gfCNCPoint2[21603] = {X 522.5718, Y 34.1930, Z -3.0000, A 0.000, B 0.000, C 0.000 }
gfCNCPoint2[21604] = {X 522.0666, Y 33.3891, Z -3.0000, A 0.000, B 0.000, C 0.000 }
gfCNCPoint2[21605] = {X 521.7531, Y 32.4929, Z -3.0000, A 0.000, B 0.000, C 0.000 }
gfCNCPoint2[21606] = {X 521.6468, Y 31.5495, Z -3.0000, A 0.000, B 0.000, C 0.000 }
gfCNCPoint2[21607] = {X 521.6468, Y 24.5714, Z -3.0000, A 0.000, B 0.000, C 0.000 }
gfCNCPoint2[21608] = {X 521.7519, Y 23.6330, Z -3.0000, A 0.000, B 0.000, C 0.000 }
gfCNCPoint2[21609] = {X 522.0622, Y 22.7411, Z -3.0000, A 0.000, B 0.000, C 0.000 }
gfCNCPoint2[21610] = {X 522.5621, Y 21.9400, Z -3.0000, A 0.000, B 0.000, C 0.000 }
gfCNCPoint2[21611] = {X 523.2270, Y 21.2694, Z -3.0000, A 0.000, B 0.000, C 0.000 }
gfCNCPoint2[21612] = {X 524.0238, Y 20.7626, Z -3.0000, A 0.000, B 0.000, C 0.000 }
gfCNCPoint2[21613] = {X 524.9130, Y 20.4448, Z -3.0000, A 0.000, B 0.000, C 0.000 }
gfCNCPoint2[21614] = {X 525.8505, Y 20.3316, Z -3.0000, A 0.000, B 0.000, C 0.000 }
gfCNCPoint2[21615] = {X 526.5687, Y 20.3316, Z -3.0000, A 0.000, B 0.000, C 0.000 }
gfCNCPoint2[21616] = {X 527.3869, Y 20.4192, Z -3.0000, A 0.000, B 0.000, C 0.000 }
gfCNCPoint2[21617] = {X 528.1727, Y 20.6632, Z -3.0000, A 0.000, B 0.000, C 0.000 }
gfCNCPoint2[21618] = {X 528.8966, Y 21.0544, Z -3.0000, A 0.000, B 0.000, C 0.000 }
gfCNCPoint2[21619] = {X 529.5313, Y 21.5780, Z -3.0000, A 0.000, B 0.000, C 0.000 }
gfCNCPoint2[21620] = {X 530.0529, Y 22.2144, Z -3.0000, A 0.000, B 0.000, C 0.000 }
gfCNCPoint2[21621] = {X 534.7119, Y 22.2147, Z -3.0000, A 0.000, B 0.000, C 0.000 }
gfCNCPoint2[21622] = {X 534.7119, Y 19.6214, Z -3.0000, A 0.000, B 0.000, C 0.000 }
gfCNCPoint2[21623] = {X 524.1494, Y 19.6210, Z -3.0000, A 0.000, B 0.000, C 0.000 }
gfCNCPoint2[21624] = {X 524.1262, Y 19.6563, Z -3.0000, A 0.000, B 0.000, C 0.000 }
gfCNCPoint2[21625] = {X 523.6036, Y 20.2891, Z -3.0000, A 0.000, B 0.000, C 0.000 }
gfCNCPoint2[21626] = {X 522.9689, Y 20.8095, Z -3.0000, A 0.000, B 0.000, C 0.000 }
gfCNCPoint2[21627] = {X 522.2458, Y 21.1978, Z -3.0000, A 0.000, B 0.000, C 0.000 }
gfCNCPoint2[21628] = {X 521.4615, Y 21.4395, Z -3.0000, A 0.000, B 0.000, C 0.000 }
gfCNCPoint2[21629] = {X 520.6453, Y 21.5256, Z -3.0000, A 0.000, B 0.000, C 0.000 }
gfCNCPoint2[21630] = {X 519.9691, Y 21.5257, Z -3.0000, A 0.000, B 0.000, C 0.000 }
gfCNCPoint2[21631] = {X 519.0256, Y 21.4194, Z -3.0000, A 0.000, B 0.000, C 0.000 }
gfCNCPoint2[21632] = {X 518.1294, Y 21.1058, Z -3.0000, A 0.000, B 0.000, C 0.000 }
gfCNCPoint2[21633] = {X 517.3255, Y 20.6007, Z -3.0000, A 0.000, B 0.000, C 0.000 }
gfCNCPoint2[21634] = {X 516.6541, Y 19.9293, Z -3.0000, A 0.000, B 0.000, C 0.000 }
gfCNCPoint2[21635] = {X 516.1490, Y 19.1254, Z -3.0000, A 0.000, B 0.000, C 0.000 }
gfCNCPoint2[21636] = {X 515.8354, Y 18.2292, Z -3.0000, A 0.000, B 0.000, C 0.000 }
gfCNCPoint2[21637] = {X 515.7291, Y 17.2857, Z -3.0000, A 0.000, B 0.000, C 0.000 }
gfCNCPoint2[21638] = {X 515.7291, Y 10.3077, Z -3.0000, A 0.000, B 0.000, C 0.000 }
gfCNCPoint2[21639] = {X 515.8342, Y 9.3696, Z -3.0000, A 0.000, B 0.000, C 0.000 }
gfCNCPoint2[21640] = {X 516.1442, Y 8.4780, Z -3.0000, A 0.000, B 0.000, C 0.000 }
gfCNCPoint2[21641] = {X 516.6438, Y 7.6771, Z -3.0000, A 0.000, B 0.000, C 0.000 }
gfCNCPoint2[21642] = {X 517.3082, Y 7.0066, Z -3.0000, A 0.000, B 0.000, C 0.000 }
gfCNCPoint2[21643] = {X 518.1045, Y 6.4997, Z -3.0000, A 0.000, B 0.000, C 0.000 }
gfCNCPoint2[21644] = {X 518.9932, Y 6.1815, Z -3.0000, A 0.000, B 0.000, C 0.000 }
gfCNCPoint2[21645] = {X 519.9303, Y 6.0679, Z -3.0000, A 0.000, B 0.000, C 0.000 }
gfCNCPoint2[21646] = {X 520.6494, Y 6.0679, Z -3.0000, A 0.000, B 0.000, C 0.000 }
gfCNCPoint2[21647] = {X 521.4680, Y 6.1552, Z -3.0000, A 0.000, B 0.000, C 0.000 }
gfCNCPoint2[21648] = {X 522.2542, Y 6.3991, Z -3.0000, A 0.000, B 0.000, C 0.000 }
gfCNCPoint2[21649] = {X 522.9784, Y 6.7903, Z -3.0000, A 0.000, B 0.000, C 0.000 }
gfCNCPoint2[21650] = {X 523.6134, Y 7.3141, Z -3.0000, A 0.000, B 0.000, C 0.000 }
gfCNCPoint2[21651] = {X 524.1353, Y 7.9507, Z -3.0000, A 0.000, B 0.000, C 0.000 }
gfCNCPoint2[21652] = {X 533.9639, Y 7.9510, Z -3.0000, A 0.000, B 0.000, C 0.000 }
gfCNCPoint2[21653] = {X 533.9640, Y 3.9510, Z -3.0000, A 0.000, B 0.000, C 0.000 }
gfCNCPoint2[21654] = {X 533.9638, Y 8.0310, Z -3.0000, A 0.000, B 0.000, C 0.000 }
gfCNCPoint2[21655] = {X 543.7521, Y 8.0312, Z -3.0000, A 0.000, B 0.000, C 0.000 }
gfCNCPoint2[21656] = {X 544.6963, Y 8.1132, Z -3.0000, A 0.000, B 0.000, C 0.000 }
gfCNCPoint2[21657] = {X 545.5976, Y 8.4064, Z -3.0000, A 0.000, B 0.000, C 0.000 }
gfCNCPoint2[21658] = {X 546.4091, Y 8.8959, Z -3.0000, A 0.000, B 0.000, C 0.000 }
gfCNCPoint2[21659] = {X 547.0891, Y 9.5561, Z -3.0000, A 0.000, B 0.000, C 0.000 }
gfCNCPoint2[21660] = {X 547.6021, Y 10.3530, Z -3.0000, A 0.000, B 0.000, C 0.000 }
gfCNCPoint2[21661] = {X 547.9218, Y 11.2452, Z -3.0000, A 0.000, B 0.000, C 0.000 }
gfCNCPoint2[21662] = {X 548.0314, Y 12.1866, Z -3.0000, A 0.000, B 0.000, C 0.000 }
gfCNCPoint2[21663] = {X 548.0312, Y 13.0208, Z -3.0000, A 0.000, B 0.000, C 0.000 }
gfCNCPoint2[21664] = {X 547.9287, Y 13.8966, Z -3.0000, A 0.000, B 0.000, C 0.000 }
gfCNCPoint2[21665] = {X 547.6440, Y 14.7310, Z -3.0000, A 0.000, B 0.000, C 0.000 }
gfCNCPoint2[21666] = {X 547.1898, Y 15.4868, Z -3.0000, A 0.000, B 0.000, C 0.000 }
gfCNCPoint2[21667] = {X 546.5866, Y 16.1298, Z -3.0000, A 0.000, B 0.000, C 0.000 }
gfCNCPoint2[21668] = {X 546.5032, Y 16.1997, Z -3.0000, A 0.000, B 0.000, C 0.000 }
gfCNCPoint2[21669] = {X 546.5034, Y 40.9897, Z -3.0000, A 0.000, B 0.000, C 0.000 }
gfCNCPoint2[21670] = {X 546.5832, Y 41.0542, Z -3.0000, A 0.000, B 0.000, C 0.000 }
gfCNCPoint2[21671] = {X 547.1891, Y 41.6991, Z -3.0000, A 0.000, B 0.000, C 0.000 }
gfCNCPoint2[21672] = {X 547.6449, Y 42.4577, Z -3.0000, A 0.000, B 0.000, C 0.000 }
gfCNCPoint2[21673] = {X 547.9299, Y 43.2955, Z -3.0000, A 0.000, B 0.000, C 0.000 }
gfCNCPoint2[21674] = {X 548.0313, Y 44.1746, Z -3.0000, A 0.000, B 0.000, C 0.000 }
gfCNCPoint2[21675] = {X 548.0314, Y 45.0003, Z -3.0000, A 0.000, B 0.000, C 0.000 }
gfCNCPoint2[21676] = {X 547.9218, Y 45.9416, Z -3.0000, A 0.000, B 0.000, C 0.000 }
gfCNCPoint2[21677] = {X 547.6021, Y 46.8338, Z -3.0000, A 0.000, B 0.000, C 0.000 }
gfCNCPoint2[21678] = {X 547.0891, Y 47.6306, Z -3.0000, A 0.000, B 0.000, C 0.000 }
gfCNCPoint2[21679] = {X 546.4091, Y 48.2908, Z -3.0000, A 0.000, B 0.000, C 0.000 }
gfCNCPoint2[21680] = {X 545.5975, Y 48.7802, Z -3.0000, A 0.000, B 0.000, C 0.000 }
gfCNCPoint2[21681] = {X 544.6963, Y 49.0734, Z -3.0000, A 0.000, B 0.000, C 0.000 }
gfCNCPoint2[21682] = {X 543.7521, Y 49.1553, Z -3.0000, A 0.000, B 0.000, C 0.000 }
gfCNCPoint2[21683] = {X 523.9613, Y 49.1558, Z -3.0000, A 0.000, B 0.000, C 0.000 }
gfCNCPoint2[21684] = {X 523.4346, Y 49.7883, Z -3.0000, A 0.000, B 0.000, C 0.000 }
gfCNCPoint2[21685] = {X 522.7974, Y 50.3095, Z -3.0000, A 0.000, B 0.000, C 0.000 }
gfCNCPoint2[21686] = {X 522.0729, Y 50.7002, Z -3.0000, A 0.000, B 0.000, C 0.000 }
gfCNCPoint2[21687] = {X 521.2874, Y 50.9464, Z -3.0000, A 0.000, B 0.000, C 0.000 }
gfCNCPoint2[21688] = {X 520.4695, Y 51.0391, Z -3.0000, A 0.000, B 0.000, C 0.000 }
gfCNCPoint2[21689] = {X 519.7998, Y 51.0391, Z -3.0000, A 0.000, B 0.000, C 0.000 }
gfCNCPoint2[21690] = {X 518.8741, Y 50.9348, Z -3.0000, A 0.000, B 0.000, C 0.000 }
gfCNCPoint2[21691] = {X 517.9948, Y 50.6272, Z -3.0000, A 0.000, B 0.000, C 0.000 }
gfCNCPoint2[21692] = {X 517.2061, Y 50.1315, Z -3.0000, A 0.000, B 0.000, C 0.000 }
gfCNCPoint2[21693] = {X 516.5474, Y 49.4728, Z -3.0000, A 0.000, B 0.000, C 0.000 }
gfCNCPoint2[21694] = {X 516.0517, Y 48.6841, Z -3.0000, A 0.000, B 0.000, C 0.000 }
gfCNCPoint2[21695] = {X 515.7441, Y 47.8048, Z -3.0000, A 0.000, B 0.000, C 0.000 }
gfCNCPoint2[21696] = {X 515.6398, Y 46.8791, Z -3.0000, A 0.000, B 0.000, C 0.000 }
gfCNCPoint2[21697] = {X 515.6398, Y 39.9011, Z -3.0000, A 0.000, B 0.000, C 0.000 }
gfCNCPoint2[21698] = {X 515.7429, Y 38.9805, Z -3.0000, A 0.000, B 0.000, C 0.000 }
gfCNCPoint2[21699] = {X 516.0472, Y 38.1056, Z -3.0000, A 0.000, B 0.000, C 0.000 }
gfCNCPoint2[21700] = {X 516.5376, Y 37.3197, Z -3.0000, A 0.000, B 0.000, C 0.000 }
gfCNCPoint2[21701] = {X 517.1897, Y 36.6618, Z -3.0000, A 0.000, B 0.000, C 0.000 }
gfCNCPoint2[21702] = {X 517.9713, Y 36.1645, Z -3.0000, A 0.000, B 0.000, C 0.000 }
gfCNCPoint2[21703] = {X 518.8435, Y 35.8525, Z -3.0000, A 0.000, B 0.000, C 0.000 }
gfCNCPoint2[21704] = {X 519.7631, Y 35.7413, Z -3.0000, A 0.000, B 0.000, C 0.000 }
gfCNCPoint2[21705] = {X 520.5247, Y 35.7415, Z -3.0000, A 0.000, B 0.000, C 0.000 }
gfCNCPoint2[21706] = {X 521.3372, Y 35.8329, Z -3.0000, A 0.000, B 0.000, C 0.000 }
gfCNCPoint2[21707] = {X 522.1162, Y 36.0815, Z -3.0000, A 0.000, B 0.000, C 0.000 }
gfCNCPoint2[21708] = {X 522.8315, Y 36.4776, Z -3.0000, A 0.000, B 0.000, C 0.000 }
gfCNCPoint2[21709] = {X 523.4555, Y 37.0060, Z -3.0000, A 0.000, B 0.000, C 0.000 }
gfCNCPoint2[21710] = {X 523.9640, Y 37.6462, Z -3.0000, A 0.000, B 0.000, C 0.000 }
gfCNCPoint2[21711] = {X 534.7919, Y 37.6467, Z -3.0000, A 0.000, B 0.000, C 0.000 }
gfCNCPoint2[21712] = {X 534.7919, Y 33.8050, Z -3.0000, A 0.000, B 0.000, C 0.000 }
gfCNCPoint2[21713] = {X 530.0216, Y 33.8045, Z -3.0000, A 0.000, B 0.000, C 0.000 }
gfCNCPoint2[21714] = {X 529.9749, Y 33.8791, Z -3.0000, A 0.000, B 0.000, C 0.000 }
gfCNCPoint2[21715] = {X 529.4624, Y 34.4985, Z -3.0000, A 0.000, B 0.000, C 0.000 }
gfCNCPoint2[21716] = {X 528.8404, Y 35.0079, Z -3.0000, A 0.000, B 0.000, C 0.000 }
gfCNCPoint2[21717] = {X 528.1319, Y 35.3880, Z -3.0000, A 0.000, B 0.000, C 0.000 }
gfCNCPoint2[21718] = {X 527.3636, Y 35.6248, Z -3.0000, A 0.000, B 0.000, C 0.000 }
gfCNCPoint2[21719] = {X 526.5641, Y 35.7093, Z -3.0000, A 0.000, B 0.000, C 0.000 }
gfCNCPoint2[21720] = {X 525.8868, Y 35.7095, Z -3.0000, A 0.000, B 0.000, C 0.000 }
gfCNCPoint2[21721] = {X 524.9611, Y 35.6052, Z -3.0000, A 0.000, B 0.000, C 0.000 }
gfCNCPoint2[21722] = {X 524.0818, Y 35.2975, Z -3.0000, A 0.000, B 0.000, C 0.000 }
gfCNCPoint2[21723] = {X 523.2930, Y 34.8019, Z -3.0000, A 0.000, B 0.000, C 0.000 }
gfCNCPoint2[21724] = {X 522.6343, Y 34.1432, Z -3.0000, A 0.000, B 0.000, C 0.000 }
gfCNCPoint2[21725] = {X 522.1387, Y 33.3544, Z -3.0000, A 0.000, B 0.000, C 0.000 }
gfCNCPoint2[21726] = {X 521.8311, Y 32.4751, Z -3.0000, A 0.000, B 0.000, C 0.000 }
gfCNCPoint2[21727] = {X 521.7268, Y 31.5495, Z -3.0000, A 0.000, B 0.000, C 0.000 }
gfCNCPoint2[21728] = {X 521.7268, Y 24.5714, Z -3.0000, A 0.000, B 0.000, C 0.000 }
gfCNCPoint2[21729] = {X 521.8299, Y 23.6507, Z -3.0000, A 0.000, B 0.000, C 0.000 }
gfCNCPoint2[21730] = {X 522.1343, Y 22.7756, Z -3.0000, A 0.000, B 0.000, C 0.000 }
gfCNCPoint2[21731] = {X 522.6248, Y 21.9897, Z -3.0000, A 0.000, B 0.000, C 0.000 }
gfCNCPoint2[21732] = {X 523.2772, Y 21.3317, Z -3.0000, A 0.000, B 0.000, C 0.000 }
gfCNCPoint2[21733] = {X 524.0589, Y 20.8345, Z -3.0000, A 0.000, B 0.000, C 0.000 }
gfCNCPoint2[21734] = {X 524.9313, Y 20.5226, Z -3.0000, A 0.000, B 0.000, C 0.000 }
gfCNCPoint2[21735] = {X 525.8511, Y 20.4116, Z -3.0000, A 0.000, B 0.000, C 0.000 }
gfCNCPoint2[21736] = {X 526.5679, Y 20.4116, Z -3.0000, A 0.000, B 0.000, C 0.000 }
gfCNCPoint2[21737] = {X 527.3790, Y 20.4993, Z -3.0000, A 0.000, B 0.000, C 0.000 }
gfCNCPoint2[21738] = {X 528.1573, Y 20.7436, Z -3.0000, A 0.000, B 0.000, C 0.000 }
gfCNCPoint2[21739] = {X 528.8730, Y 21.1351, Z -3.0000, A 0.000, B 0.000, C 0.000 }
gfCNCPoint2[21740] = {X 529.4986, Y 21.6587, Z -3.0000, A 0.000, B 0.000, C 0.000 }
gfCNCPoint2[21741] = {X 530.0099, Y 22.2944, Z -3.0000, A 0.000, B 0.000, C 0.000 }
gfCNCPoint2[21742] = {X 534.7919, Y 22.2947, Z -3.0000, A 0.000, B 0.000, C 0.000 }
gfCNCPoint2[21743] = {X 534.7919, Y 19.5414, Z -3.0000, A 0.000, B 0.000, C 0.000 }
gfCNCPoint2[21744] = {X 524.1051, Y 19.5410, Z -3.0000, A 0.000, B 0.000, C 0.000 }
gfCNCPoint2[21745] = {X 524.0765, Y 19.5866, Z -3.0000, A 0.000, B 0.000, C 0.000 }
gfCNCPoint2[21746] = {X 523.5641, Y 20.2155, Z -3.0000, A 0.000, B 0.000, C 0.000 }
gfCNCPoint2[21747] = {X 522.9393, Y 20.7329, Z -3.0000, A 0.000, B 0.000, C 0.000 }
gfCNCPoint2[21748] = {X 522.2260, Y 21.1193, Z -3.0000, A 0.000, B 0.000, C 0.000 }
gfCNCPoint2[21749] = {X 521.4513, Y 21.3599, Z -3.0000, A 0.000, B 0.000, C 0.000 }
gfCNCPoint2[21750] = {X 520.6447, Y 21.4456, Z -3.0000, A 0.000, B 0.000, C 0.000 }
gfCNCPoint2[21751] = {X 519.9691, Y 21.4457, Z -3.0000, A 0.000, B 0.000, C 0.000 }
gfCNCPoint2[21752] = {X 519.0434, Y 21.3414, Z -3.0000, A 0.000, B 0.000, C 0.000 }
gfCNCPoint2[21753] = {X 518.1641, Y 21.0337, Z -3.0000, A 0.000, B 0.000, C 0.000 }
gfCNCPoint2[21754] = {X 517.3754, Y 20.5381, Z -3.0000, A 0.000, B 0.000, C 0.000 }
gfCNCPoint2[21755] = {X 516.7167, Y 19.8794, Z -3.0000, A 0.000, B 0.000, C 0.000 }
gfCNCPoint2[21756] = {X 516.2211, Y 19.0907, Z -3.0000, A 0.000, B 0.000, C 0.000 }
gfCNCPoint2[21757] = {X 515.9134, Y 18.2114, Z -3.0000, A 0.000, B 0.000, C 0.000 }
gfCNCPoint2[21758] = {X 515.8091, Y 17.2857, Z -3.0000, A 0.000, B 0.000, C 0.000 }
gfCNCPoint2[21759] = {X 515.8091, Y 10.3077, Z -3.0000, A 0.000, B 0.000, C 0.000 }
gfCNCPoint2[21760] = {X 515.9122, Y 9.3873, Z -3.0000, A 0.000, B 0.000, C 0.000 }
gfCNCPoint2[21761] = {X 516.2164, Y 8.5125, Z -3.0000, A 0.000, B 0.000, C 0.000 }
gfCNCPoint2[21762] = {X 516.7065, Y 7.7267, Z -3.0000, A 0.000, B 0.000, C 0.000 }
gfCNCPoint2[21763] = {X 517.3584, Y 7.0689, Z -3.0000, A 0.000, B 0.000, C 0.000 }
gfCNCPoint2[21764] = {X 518.1397, Y 6.5715, Z -3.0000, A 0.000, B 0.000, C 0.000 }
gfCNCPoint2[21765] = {X 519.0117, Y 6.2594, Z -3.0000, A 0.000, B 0.000, C 0.000 }
gfCNCPoint2[21766] = {X 519.9311, Y 6.1479, Z -3.0000, A 0.000, B 0.000, C 0.000 }
gfCNCPoint2[21767] = {X 520.6487, Y 6.1479, Z -3.0000, A 0.000, B 0.000, C 0.000 }
gfCNCPoint2[21768] = {X 521.4601, Y 6.2353, Z -3.0000, A 0.000, B 0.000, C 0.000 }
gfCNCPoint2[21769] = {X 522.2388, Y 6.4795, Z -3.0000, A 0.000, B 0.000, C 0.000 }
gfCNCPoint2[21770] = {X 522.9549, Y 6.8710, Z -3.0000, A 0.000, B 0.000, C 0.000 }
gfCNCPoint2[21771] = {X 523.5807, Y 7.3948, Z -3.0000, A 0.000, B 0.000, C 0.000 }
gfCNCPoint2[21772] = {X 524.0923, Y 8.0307, Z -3.0000, A 0.000, B 0.000, C 0.000 }
gfCNCPoint2[21773] = {X 533.9638, Y 8.0310, Z -3.0000, A 0.000, B 0.000, C 0.000 }
gfCNCPoint2[21774] = {X 533.9640, Y 4.0310, Z -3.0000, A 0.000, B 0.000, C 0.000 }
gfCNCPoint2[21775] = {X 533.9638, Y 8.1110, Z -3.0000, A 0.000, B 0.000, C 0.000 }
gfCNCPoint2[21776] = {X 543.7532, Y 8.1112, Z -3.0000, A 0.000, B 0.000, C 0.000 }
gfCNCPoint2[21777] = {X 544.6795, Y 8.1914, Z -3.0000, A 0.000, B 0.000, C 0.000 }
gfCNCPoint2[21778] = {X 545.5636, Y 8.4789, Z -3.0000, A 0.000, B 0.000, C 0.000 }
gfCNCPoint2[21779] = {X 546.3598, Y 8.9589, Z -3.0000, A 0.000, B 0.000, C 0.000 }
gfCNCPoint2[21780] = {X 547.0269, Y 9.6064, Z -3.0000, A 0.000, B 0.000, C 0.000 }
gfCNCPoint2[21781] = {X 547.5303, Y 10.3881, Z -3.0000, A 0.000, B 0.000, C 0.000 }
gfCNCPoint2[21782] = {X 547.8438, Y 11.2633, Z -3.0000, A 0.000, B 0.000, C 0.000 }
gfCNCPoint2[21783] = {X 547.9514, Y 12.1867, Z -3.0000, A 0.000, B 0.000, C 0.000 }
gfCNCPoint2[21784] = {X 547.9512, Y 13.0200, Z -3.0000, A 0.000, B 0.000, C 0.000 }
gfCNCPoint2[21785] = {X 547.8507, Y 13.8789, Z -3.0000, A 0.000, B 0.000, C 0.000 }
gfCNCPoint2[21786] = {X 547.5715, Y 14.6973, Z -3.0000, A 0.000, B 0.000, C 0.000 }
gfCNCPoint2[21787] = {X 547.1260, Y 15.4385, Z -3.0000, A 0.000, B 0.000, C 0.000 }
gfCNCPoint2[21788] = {X 546.5344, Y 16.0692, Z -3.0000, A 0.000, B 0.000, C 0.000 }
gfCNCPoint2[21789] = {X 546.4798, Y 16.1154, Z -3.0000, A 0.000, B 0.000, C 0.000 }
gfCNCPoint2[21790] = {X 546.4244, Y 16.1606, Z -3.0000, A 0.000, B 0.000, C 0.000 }
gfCNCPoint2[21791] = {X 546.4234, Y 41.0279, Z -3.0000, A 0.000, B 0.000, C 0.000 }
gfCNCPoint2[21792] = {X 546.5320, Y 41.1156, Z -3.0000, A 0.000, B 0.000, C 0.000 }
gfCNCPoint2[21793] = {X 547.1259, Y 41.7481, Z -3.0000, A 0.000, B 0.000, C 0.000 }
gfCNCPoint2[21794] = {X 547.5726, Y 42.4919, Z -3.0000, A 0.000, B 0.000, C 0.000 }
gfCNCPoint2[21795] = {X 547.8520, Y 43.3133, Z -3.0000, A 0.000, B 0.000, C 0.000 }
gfCNCPoint2[21796] = {X 547.9513, Y 44.1753, Z -3.0000, A 0.000, B 0.000, C 0.000 }
gfCNCPoint2[21797] = {X 547.9514, Y 45.0001, Z -3.0000, A 0.000, B 0.000, C 0.000 }
gfCNCPoint2[21798] = {X 547.8439, Y 45.9235, Z -3.0000, A 0.000, B 0.000, C 0.000 }
gfCNCPoint2[21799] = {X 547.5303, Y 46.7987, Z -3.0000, A 0.000, B 0.000, C 0.000 }
gfCNCPoint2[21800] = {X 547.0269, Y 47.5803, Z -3.0000, A 0.000, B 0.000, C 0.000 }
gfCNCPoint2[21801] = {X 546.3598, Y 48.2279, Z -3.0000, A 0.000, B 0.000, C 0.000 }
gfCNCPoint2[21802] = {X 545.5636, Y 48.7078, Z -3.0000, A 0.000, B 0.000, C 0.000 }
gfCNCPoint2[21803] = {X 544.6795, Y 48.9952, Z -3.0000, A 0.000, B 0.000, C 0.000 }
gfCNCPoint2[21804] = {X 543.7532, Y 49.0753, Z -3.0000, A 0.000, B 0.000, C 0.000 }
gfCNCPoint2[21805] = {X 523.9188, Y 49.0758, Z -3.0000, A 0.000, B 0.000, C 0.000 }
gfCNCPoint2[21806] = {X 523.4022, Y 49.7076, Z -3.0000, A 0.000, B 0.000, C 0.000 }
gfCNCPoint2[21807] = {X 522.7741, Y 50.2287, Z -3.0000, A 0.000, B 0.000, C 0.000 }
gfCNCPoint2[21808] = {X 522.0577, Y 50.6198, Z -3.0000, A 0.000, B 0.000, C 0.000 }
gfCNCPoint2[21809] = {X 521.2797, Y 50.8663, Z -3.0000, A 0.000, B 0.000, C 0.000 }
gfCNCPoint2[21810] = {X 520.4688, Y 50.9591, Z -3.0000, A 0.000, B 0.000, C 0.000 }
gfCNCPoint2[21811] = {X 519.7998, Y 50.9591, Z -3.0000, A 0.000, B 0.000, C 0.000 }
gfCNCPoint2[21812] = {X 518.8919, Y 50.8568, Z -3.0000, A 0.000, B 0.000, C 0.000 }
gfCNCPoint2[21813] = {X 518.0295, Y 50.5551, Z -3.0000, A 0.000, B 0.000, C 0.000 }
gfCNCPoint2[21814] = {X 517.2559, Y 50.0690, Z -3.0000, A 0.000, B 0.000, C 0.000 }
gfCNCPoint2[21815] = {X 516.6099, Y 49.4230, Z -3.0000, A 0.000, B 0.000, C 0.000 }
gfCNCPoint2[21816] = {X 516.1238, Y 48.6494, Z -3.0000, A 0.000, B 0.000, C 0.000 }
gfCNCPoint2[21817] = {X 515.8221, Y 47.7870, Z -3.0000, A 0.000, B 0.000, C 0.000 }
gfCNCPoint2[21818] = {X 515.7198, Y 46.8791, Z -3.0000, A 0.000, B 0.000, C 0.000 }
gfCNCPoint2[21819] = {X 515.7198, Y 39.9011, Z -3.0000, A 0.000, B 0.000, C 0.000 }
gfCNCPoint2[21820] = {X 515.8209, Y 38.9982, Z -3.0000, A 0.000, B 0.000, C 0.000 }
gfCNCPoint2[21821] = {X 516.1194, Y 38.1401, Z -3.0000, A 0.000, B 0.000, C 0.000 }
gfCNCPoint2[21822] = {X 516.6003, Y 37.3693, Z -3.0000, A 0.000, B 0.000, C 0.000 }
gfCNCPoint2[21823] = {X 517.2399, Y 36.7241, Z -3.0000, A 0.000, B 0.000, C 0.000 }
gfCNCPoint2[21824] = {X 518.0064, Y 36.2364, Z -3.0000, A 0.000, B 0.000, C 0.000 }
gfCNCPoint2[21825] = {X 518.8619, Y 35.9304, Z -3.0000, A 0.000, B 0.000, C 0.000 }
gfCNCPoint2[21826] = {X 519.7638, Y 35.8213, Z -3.0000, A 0.000, B 0.000, C 0.000 }
gfCNCPoint2[21827] = {X 520.5236, Y 35.8215, Z -3.0000, A 0.000, B 0.000, C 0.000 }
gfCNCPoint2[21828] = {X 521.3290, Y 35.9129, Z -3.0000, A 0.000, B 0.000, C 0.000 }
gfCNCPoint2[21829] = {X 522.1004, Y 36.1618, Z -3.0000, A 0.000, B 0.000, C 0.000 }
gfCNCPoint2[21830] = {X 522.8074, Y 36.5583, Z -3.0000, A 0.000, B 0.000, C 0.000 }
gfCNCPoint2[21831] = {X 523.4221, Y 37.0867, Z -3.0000, A 0.000, B 0.000, C 0.000 }
gfCNCPoint2[21832] = {X 523.9202, Y 37.7262, Z -3.0000, A 0.000, B 0.000, C 0.000 }
gfCNCPoint2[21833] = {X 534.8719, Y 37.7267, Z -3.0000, A 0.000, B 0.000, C 0.000 }
gfCNCPoint2[21834] = {X 534.8719, Y 33.7250, Z -3.0000, A 0.000, B 0.000, C 0.000 }
gfCNCPoint2[21835] = {X 529.9773, Y 33.7245, Z -3.0000, A 0.000, B 0.000, C 0.000 }
gfCNCPoint2[21836] = {X 529.9071, Y 33.8366, Z -3.0000, A 0.000, B 0.000, C 0.000 }
gfCNCPoint2[21837] = {X 529.2612, Y 34.5790, Z -3.0000, A 0.000, B 0.000, C 0.000 }
gfCNCPoint2[21838] = {X 528.4563, Y 35.1452, Z -3.0000, A 0.000, B 0.000, C 0.000 }
gfCNCPoint2[21839] = {X 527.5392, Y 35.5023, Z -3.0000, A 0.000, B 0.000, C 0.000 }
gfCNCPoint2[21840] = {X 526.5634, Y 35.6293, Z -3.0000, A 0.000, B 0.000, C 0.000 }
gfCNCPoint2[21841] = {X 525.8868, Y 35.6295, Z -3.0000, A 0.000, B 0.000, C 0.000 }
gfCNCPoint2[21842] = {X 524.9789, Y 35.5272, Z -3.0000, A 0.000, B 0.000, C 0.000 }
gfCNCPoint2[21843] = {X 524.1165, Y 35.2254, Z -3.0000, A 0.000, B 0.000, C 0.000 }
gfCNCPoint2[21844] = {X 523.3429, Y 34.7393, Z -3.0000, A 0.000, B 0.000, C 0.000 }
gfCNCPoint2[21845] = {X 522.6969, Y 34.0933, Z -3.0000, A 0.000, B 0.000, C 0.000 }
gfCNCPoint2[21846] = {X 522.2108, Y 33.3197, Z -3.0000, A 0.000, B 0.000, C 0.000 }
gfCNCPoint2[21847] = {X 521.9091, Y 32.4573, Z -3.0000, A 0.000, B 0.000, C 0.000 }
gfCNCPoint2[21848] = {X 521.8068, Y 31.5495, Z -3.0000, A 0.000, B 0.000, C 0.000 }
gfCNCPoint2[21849] = {X 521.8068, Y 24.5714, Z -3.0000, A 0.000, B 0.000, C 0.000 }
gfCNCPoint2[21850] = {X 521.9079, Y 23.6684, Z -3.0000, A 0.000, B 0.000, C 0.000 }
gfCNCPoint2[21851] = {X 522.2065, Y 22.8102, Z -3.0000, A 0.000, B 0.000, C 0.000 }
gfCNCPoint2[21852] = {X 522.6876, Y 22.0393, Z -3.0000, A 0.000, B 0.000, C 0.000 }
gfCNCPoint2[21853] = {X 523.3273, Y 21.3940, Z -3.0000, A 0.000, B 0.000, C 0.000 }
gfCNCPoint2[21854] = {X 524.0941, Y 20.9064, Z -3.0000, A 0.000, B 0.000, C 0.000 }
gfCNCPoint2[21855] = {X 524.9497, Y 20.6005, Z -3.0000, A 0.000, B 0.000, C 0.000 }
gfCNCPoint2[21856] = {X 525.8518, Y 20.4916, Z -3.0000, A 0.000, B 0.000, C 0.000 }
gfCNCPoint2[21857] = {X 526.5672, Y 20.4916, Z -3.0000, A 0.000, B 0.000, C 0.000 }
gfCNCPoint2[21858] = {X 527.3711, Y 20.5794, Z -3.0000, A 0.000, B 0.000, C 0.000 }
gfCNCPoint2[21859] = {X 528.1419, Y 20.8240, Z -3.0000, A 0.000, B 0.000, C 0.000 }
gfCNCPoint2[21860] = {X 528.8493, Y 21.2158, Z -3.0000, A 0.000, B 0.000, C 0.000 }
gfCNCPoint2[21861] = {X 529.4655, Y 21.7395, Z -3.0000, A 0.000, B 0.000, C 0.000 }
gfCNCPoint2[21862] = {X 529.9664, Y 22.3744, Z -3.0000, A 0.000, B 0.000, C 0.000 }
gfCNCPoint2[21863] = {X 534.8719, Y 22.3747, Z -3.0000, A 0.000, B 0.000, C 0.000 }
gfCNCPoint2[21864] = {X 534.8719, Y 19.4614, Z -3.0000, A 0.000, B 0.000, C 0.000 }
gfCNCPoint2[21865] = {X 524.0608, Y 19.4610, Z -3.0000, A 0.000, B 0.000, C 0.000 }
gfCNCPoint2[21866] = {X 524.0087, Y 19.5442, Z -3.0000, A 0.000, B 0.000, C 0.000 }
gfCNCPoint2[21867] = {X 523.5061, Y 20.1604, Z -3.0000, A 0.000, B 0.000, C 0.000 }
gfCNCPoint2[21868] = {X 522.8935, Y 20.6674, Z -3.0000, A 0.000, B 0.000, C 0.000 }
gfCNCPoint2[21869] = {X 522.1942, Y 21.0459, Z -3.0000, A 0.000, B 0.000, C 0.000 }
gfCNCPoint2[21870] = {X 521.4348, Y 21.2816, Z -3.0000, A 0.000, B 0.000, C 0.000 }
gfCNCPoint2[21871] = {X 520.6440, Y 21.3656, Z -3.0000, A 0.000, B 0.000, C 0.000 }
gfCNCPoint2[21872] = {X 519.9691, Y 21.3657, Z -3.0000, A 0.000, B 0.000, C 0.000 }
gfCNCPoint2[21873] = {X 519.0612, Y 21.2634, Z -3.0000, A 0.000, B 0.000, C 0.000 }
gfCNCPoint2[21874] = {X 518.1989, Y 20.9617, Z -3.0000, A 0.000, B 0.000, C 0.000 }
gfCNCPoint2[21875] = {X 517.4253, Y 20.4756, Z -3.0000, A 0.000, B 0.000, C 0.000 }
gfCNCPoint2[21876] = {X 516.7792, Y 19.8296, Z -3.0000, A 0.000, B 0.000, C 0.000 }
gfCNCPoint2[21877] = {X 516.2932, Y 19.0560, Z -3.0000, A 0.000, B 0.000, C 0.000 }
gfCNCPoint2[21878] = {X 515.9914, Y 18.1936, Z -3.0000, A 0.000, B 0.000, C 0.000 }
gfCNCPoint2[21879] = {X 515.8891, Y 17.2857, Z -3.0000, A 0.000, B 0.000, C 0.000 }
gfCNCPoint2[21880] = {X 515.8891, Y 10.3077, Z -3.0000, A 0.000, B 0.000, C 0.000 }
gfCNCPoint2[21881] = {X 515.9902, Y 9.4050, Z -3.0000, A 0.000, B 0.000, C 0.000 }
gfCNCPoint2[21882] = {X 516.2885, Y 8.5471, Z -3.0000, A 0.000, B 0.000, C 0.000 }
gfCNCPoint2[21883] = {X 516.7693, Y 7.7764, Z -3.0000, A 0.000, B 0.000, C 0.000 }
gfCNCPoint2[21884] = {X 517.4086, Y 7.1312, Z -3.0000, A 0.000, B 0.000, C 0.000 }
gfCNCPoint2[21885] = {X 518.1749, Y 6.6434, Z -3.0000, A 0.000, B 0.000, C 0.000 }
gfCNCPoint2[21886] = {X 519.0301, Y 6.3372, Z -3.0000, A 0.000, B 0.000, C 0.000 }
gfCNCPoint2[21887] = {X 519.9318, Y 6.2279, Z -3.0000, A 0.000, B 0.000, C 0.000 }
gfCNCPoint2[21888] = {X 520.6480, Y 6.2279, Z -3.0000, A 0.000, B 0.000, C 0.000 }
gfCNCPoint2[21889] = {X 521.4522, Y 6.3154, Z -3.0000, A 0.000, B 0.000, C 0.000 }
gfCNCPoint2[21890] = {X 522.2234, Y 6.5599, Z -3.0000, A 0.000, B 0.000, C 0.000 }
gfCNCPoint2[21891] = {X 522.9312, Y 6.9518, Z -3.0000, A 0.000, B 0.000, C 0.000 }
gfCNCPoint2[21892] = {X 523.5477, Y 7.4756, Z -3.0000, A 0.000, B 0.000, C 0.000 }
gfCNCPoint2[21893] = {X 524.0487, Y 8.1107, Z -3.0000, A 0.000, B 0.000, C 0.000 }
gfCNCPoint2[21894] = {X 533.9638, Y 8.1110, Z -3.0000, A 0.000, B 0.000, C 0.000 }
gfCNCPoint2[21895] = {X 533.9640, Y 4.1110, Z -3.0000, A 0.000, B 0.000, C 0.000 }
gfCNCPoint2[21896] = {X 533.9638, Y 8.1910, Z -3.0000, A 0.000, B 0.000, C 0.000 }
gfCNCPoint2[21897] = {X 543.7544, Y 8.1912, Z -3.0000, A 0.000, B 0.000, C 0.000 }
gfCNCPoint2[21898] = {X 544.6626, Y 8.2696, Z -3.0000, A 0.000, B 0.000, C 0.000 }
gfCNCPoint2[21899] = {X 545.5296, Y 8.5513, Z -3.0000, A 0.000, B 0.000, C 0.000 }
gfCNCPoint2[21900] = {X 546.3105, Y 9.0218, Z -3.0000, A 0.000, B 0.000, C 0.000 }
gfCNCPoint2[21901] = {X 546.9647, Y 9.6567, Z -3.0000, A 0.000, B 0.000, C 0.000 }
gfCNCPoint2[21902] = {X 547.4584, Y 10.4232, Z -3.0000, A 0.000, B 0.000, C 0.000 }
gfCNCPoint2[21903] = {X 547.7659, Y 11.2814, Z -3.0000, A 0.000, B 0.000, C 0.000 }
gfCNCPoint2[21904] = {X 547.8714, Y 12.1869, Z -3.0000, A 0.000, B 0.000, C 0.000 }
gfCNCPoint2[21905] = {X 547.8712, Y 13.0192, Z -3.0000, A 0.000, B 0.000, C 0.000 }
gfCNCPoint2[21906] = {X 547.7727, Y 13.8612, Z -3.0000, A 0.000, B 0.000, C 0.000 }
gfCNCPoint2[21907] = {X 547.4989, Y 14.6636, Z -3.0000, A 0.000, B 0.000, C 0.000 }
gfCNCPoint2[21908] = {X 547.0622, Y 15.3903, Z -3.0000, A 0.000, B 0.000, C 0.000 }
gfCNCPoint2[21909] = {X 546.4821, Y 16.0086, Z -3.0000, A 0.000, B 0.000, C 0.000 }
gfCNCPoint2[21910] = {X 546.4146, Y 16.0655, Z -3.0000, A 0.000, B 0.000, C 0.000 }
gfCNCPoint2[21911] = {X 546.3458, Y 16.1209, Z -3.0000, A 0.000, B 0.000, C 0.000 }
gfCNCPoint2[21912] = {X 546.3432, Y 16.3116, Z -3.0000, A 0.000, B 0.000, C 0.000 }
gfCNCPoint2[21913] = {X 546.3434, Y 41.0661, Z -3.0000, A 0.000, B 0.000, C 0.000 }
gfCNCPoint2[21914] = {X 546.4824, Y 41.1784, Z -3.0000, A 0.000, B 0.000, C 0.000 }
gfCNCPoint2[21915] = {X 547.0685, Y 41.8049, Z -3.0000, A 0.000, B 0.000, C 0.000 }
gfCNCPoint2[21916] = {X 547.5076, Y 42.5421, Z -3.0000, A 0.000, B 0.000, C 0.000 }
gfCNCPoint2[21917] = {X 547.7794, Y 43.3559, Z -3.0000, A 0.000, B 0.000, C 0.000 }
gfCNCPoint2[21918] = {X 547.8714, Y 44.2089, Z -3.0000, A 0.000, B 0.000, C 0.000 }
gfCNCPoint2[21919] = {X 547.8714, Y 45.0000, Z -3.0000, A 0.000, B 0.000, C 0.000 }
gfCNCPoint2[21920] = {X 547.7659, Y 45.9054, Z -3.0000, A 0.000, B 0.000, C 0.000 }
gfCNCPoint2[21921] = {X 547.4584, Y 46.7636, Z -3.0000, A 0.000, B 0.000, C 0.000 }
gfCNCPoint2[21922] = {X 546.9647, Y 47.5300, Z -3.0000, A 0.000, B 0.000, C 0.000 }
gfCNCPoint2[21923] = {X 546.3105, Y 48.1649, Z -3.0000, A 0.000, B 0.000, C 0.000 }
gfCNCPoint2[21924] = {X 545.5296, Y 48.6353, Z -3.0000, A 0.000, B 0.000, C 0.000 }
gfCNCPoint2[21925] = {X 544.6626, Y 48.9170, Z -3.0000, A 0.000, B 0.000, C 0.000 }
gfCNCPoint2[21926] = {X 543.7544, Y 48.9953, Z -3.0000, A 0.000, B 0.000, C 0.000 }
gfCNCPoint2[21927] = {X 523.8758, Y 48.9958, Z -3.0000, A 0.000, B 0.000, C 0.000 }
gfCNCPoint2[21928] = {X 523.3694, Y 49.6269, Z -3.0000, A 0.000, B 0.000, C 0.000 }
gfCNCPoint2[21929] = {X 522.7505, Y 50.1479, Z -3.0000, A 0.000, B 0.000, C 0.000 }
gfCNCPoint2[21930] = {X 522.0424, Y 50.5393, Z -3.0000, A 0.000, B 0.000, C 0.000 }
gfCNCPoint2[21931] = {X 521.2718, Y 50.7862, Z -3.0000, A 0.000, B 0.000, C 0.000 }
gfCNCPoint2[21932] = {X 520.4681, Y 50.8791, Z -3.0000, A 0.000, B 0.000, C 0.000 }
gfCNCPoint2[21933] = {X 519.7998, Y 50.8791, Z -3.0000, A 0.000, B 0.000, C 0.000 }
gfCNCPoint2[21934] = {X 518.9097, Y 50.7788, Z -3.0000, A 0.000, B 0.000, C 0.000 }
gfCNCPoint2[21935] = {X 518.0642, Y 50.4830, Z -3.0000, A 0.000, B 0.000, C 0.000 }
gfCNCPoint2[21936] = {X 517.3058, Y 50.0064, Z -3.0000, A 0.000, B 0.000, C 0.000 }
gfCNCPoint2[21937] = {X 516.6724, Y 49.3731, Z -3.0000, A 0.000, B 0.000, C 0.000 }
gfCNCPoint2[21938] = {X 516.1959, Y 48.6147, Z -3.0000, A 0.000, B 0.000, C 0.000 }
gfCNCPoint2[21939] = {X 515.9001, Y 47.7692, Z -3.0000, A 0.000, B 0.000, C 0.000 }
gfCNCPoint2[21940] = {X 515.7998, Y 46.8791, Z -3.0000, A 0.000, B 0.000, C 0.000 }
gfCNCPoint2[21941] = {X 515.7998, Y 39.9011, Z -3.0000, A 0.000, B 0.000, C 0.000 }
gfCNCPoint2[21942] = {X 515.9001, Y 39.0110, Z -3.0000, A 0.000, B 0.000, C 0.000 }
gfCNCPoint2[21943] = {X 516.1959, Y 38.1655, Z -3.0000, A 0.000, B 0.000, C 0.000 }
gfCNCPoint2[21944] = {X 516.6725, Y 37.4071, Z -3.0000, A 0.000, B 0.000, C 0.000 }
gfCNCPoint2[21945] = {X 517.3059, Y 36.7737, Z -3.0000, A 0.000, B 0.000, C 0.000 }
gfCNCPoint2[21946] = {X 518.0643, Y 36.2972, Z -3.0000, A 0.000, B 0.000, C 0.000 }
gfCNCPoint2[21947] = {X 518.9098, Y 36.0014, Z -3.0000, A 0.000, B 0.000, C 0.000 }
gfCNCPoint2[21948] = {X 519.7999, Y 35.9011, Z -3.0000, A 0.000, B 0.000, C 0.000 }
gfCNCPoint2[21949] = {X 520.5225, Y 35.9015, Z -3.0000, A 0.000, B 0.000, C 0.000 }
gfCNCPoint2[21950] = {X 521.3207, Y 35.9930, Z -3.0000, A 0.000, B 0.000, C 0.000 }
gfCNCPoint2[21951] = {X 522.0845, Y 36.2422, Z -3.0000, A 0.000, B 0.000, C 0.000 }
gfCNCPoint2[21952] = {X 522.7831, Y 36.6390, Z -3.0000, A 0.000, B 0.000, C 0.000 }
gfCNCPoint2[21953] = {X 523.3883, Y 37.1675, Z -3.0000, A 0.000, B 0.000, C 0.000 }
gfCNCPoint2[21954] = {X 523.8757, Y 37.8062, Z -3.0000, A 0.000, B 0.000, C 0.000 }
gfCNCPoint2[21955] = {X 534.9519, Y 37.8068, Z -3.0000, A 0.000, B 0.000, C 0.000 }
gfCNCPoint2[21956] = {X 534.9519, Y 34.0450, Z -3.0000, A 0.000, B 0.000, C 0.000 }
gfCNCPoint2[21957] = {X 534.9528, Y 33.6450, Z -3.0000, A 0.000, B 0.000, C 0.000 }
gfCNCPoint2[21958] = {X 529.9330, Y 33.6445, Z -3.0000, A 0.000, B 0.000, C 0.000 }
gfCNCPoint2[21959] = {X 529.8231, Y 33.8177, Z -3.0000, A 0.000, B 0.000, C 0.000 }
gfCNCPoint2[21960] = {X 529.1836, Y 34.5411, Z -3.0000, A 0.000, B 0.000, C 0.000 }
gfCNCPoint2[21961] = {X 528.3894, Y 35.0902, Z -3.0000, A 0.000, B 0.000, C 0.000 }
gfCNCPoint2[21962] = {X 527.4868, Y 35.4330, Z -3.0000, A 0.000, B 0.000, C 0.000 }
gfCNCPoint2[21963] = {X 526.5283, Y 35.5495, Z -3.0000, A 0.000, B 0.000, C 0.000 }
gfCNCPoint2[21964] = {X 525.8868, Y 35.5495, Z -3.0000, A 0.000, B 0.000, C 0.000 }
gfCNCPoint2[21965] = {X 524.9967, Y 35.4492, Z -3.0000, A 0.000, B 0.000, C 0.000 }
gfCNCPoint2[21966] = {X 524.1512, Y 35.1533, Z -3.0000, A 0.000, B 0.000, C 0.000 }
gfCNCPoint2[21967] = {X 523.3928, Y 34.6768, Z -3.0000, A 0.000, B 0.000, C 0.000 }
gfCNCPoint2[21968] = {X 522.7594, Y 34.0434, Z -3.0000, A 0.000, B 0.000, C 0.000 }
gfCNCPoint2[21969] = {X 522.2829, Y 33.2850, Z -3.0000, A 0.000, B 0.000, C 0.000 }
gfCNCPoint2[21970] = {X 521.9870, Y 32.4395, Z -3.0000, A 0.000, B 0.000, C 0.000 }
gfCNCPoint2[21971] = {X 521.8868, Y 31.5495, Z -3.0000, A 0.000, B 0.000, C 0.000 }
gfCNCPoint2[21972] = {X 521.8868, Y 24.5714, Z -3.0000, A 0.000, B 0.000, C 0.000 }
gfCNCPoint2[21973] = {X 521.9870, Y 23.6813, Z -3.0000, A 0.000, B 0.000, C 0.000 }
gfCNCPoint2[21974] = {X 522.2829, Y 22.8359, Z -3.0000, A 0.000, B 0.000, C 0.000 }
gfCNCPoint2[21975] = {X 522.7594, Y 22.0775, Z -3.0000, A 0.000, B 0.000, C 0.000 }
gfCNCPoint2[21976] = {X 523.3928, Y 21.4441, Z -3.0000, A 0.000, B 0.000, C 0.000 }
gfCNCPoint2[21977] = {X 524.1512, Y 20.9675, Z -3.0000, A 0.000, B 0.000, C 0.000 }
gfCNCPoint2[21978] = {X 524.9967, Y 20.6717, Z -3.0000, A 0.000, B 0.000, C 0.000 }
gfCNCPoint2[21979] = {X 525.8868, Y 20.5714, Z -3.0000, A 0.000, B 0.000, C 0.000 }
gfCNCPoint2[21980] = {X 526.5664, Y 20.5716, Z -3.0000, A 0.000, B 0.000, C 0.000 }
gfCNCPoint2[21981] = {X 527.3631, Y 20.6595, Z -3.0000, A 0.000, B 0.000, C 0.000 }
gfCNCPoint2[21982] = {X 528.1263, Y 20.9044, Z -3.0000, A 0.000, B 0.000, C 0.000 }
gfCNCPoint2[21983] = {X 528.8253, Y 21.2966, Z -3.0000, A 0.000, B 0.000, C 0.000 }
gfCNCPoint2[21984] = {X 529.4321, Y 21.8203, Z -3.0000, A 0.000, B 0.000, C 0.000 }
gfCNCPoint2[21985] = {X 529.9223, Y 22.4544, Z -3.0000, A 0.000, B 0.000, C 0.000 }
gfCNCPoint2[21986] = {X 534.9519, Y 22.4547, Z -3.0000, A 0.000, B 0.000, C 0.000 }
gfCNCPoint2[21987] = {X 534.9519, Y 19.7814, Z -3.0000, A 0.000, B 0.000, C 0.000 }
gfCNCPoint2[21988] = {X 534.9529, Y 19.3814, Z -3.0000, A 0.000, B 0.000, C 0.000 }
gfCNCPoint2[21989] = {X 524.0164, Y 19.3810, Z -3.0000, A 0.000, B 0.000, C 0.000 }
gfCNCPoint2[21990] = {X 523.9053, Y 19.5542, Z -3.0000, A 0.000, B 0.000, C 0.000 }
gfCNCPoint2[21991] = {X 523.2659, Y 20.2775, Z -3.0000, A 0.000, B 0.000, C 0.000 }
gfCNCPoint2[21992] = {X 522.4717, Y 20.8265, Z -3.0000, A 0.000, B 0.000, C 0.000 }
gfCNCPoint2[21993] = {X 521.5691, Y 21.1692, Z -3.0000, A 0.000, B 0.000, C 0.000 }
gfCNCPoint2[21994] = {X 520.6107, Y 21.2857, Z -3.0000, A 0.000, B 0.000, C 0.000 }
gfCNCPoint2[21995] = {X 519.9691, Y 21.2857, Z -3.0000, A 0.000, B 0.000, C 0.000 }
gfCNCPoint2[21996] = {X 519.0790, Y 21.1854, Z -3.0000, A 0.000, B 0.000, C 0.000 }
gfCNCPoint2[21997] = {X 518.2336, Y 20.8896, Z -3.0000, A 0.000, B 0.000, C 0.000 }
gfCNCPoint2[21998] = {X 517.4751, Y 20.4130, Z -3.0000, A 0.000, B 0.000, C 0.000 }
gfCNCPoint2[21999] = {X 516.8418, Y 19.7797, Z -3.0000, A 0.000, B 0.000, C 0.000 }
gfCNCPoint2[22000] = {X 516.3652, Y 19.0212, Z -3.0000, A 0.000, B 0.000, C 0.000 }
gfCNCPoint2[22001] = {X 516.0694, Y 18.1758, Z -3.0000, A 0.000, B 0.000, C 0.000 }
gfCNCPoint2[22002] = {X 515.9691, Y 17.2857, Z -3.0000, A 0.000, B 0.000, C 0.000 }
gfCNCPoint2[22003] = {X 515.9691, Y 10.3077, Z -3.0000, A 0.000, B 0.000, C 0.000 }
gfCNCPoint2[22004] = {X 516.0694, Y 9.4176, Z -3.0000, A 0.000, B 0.000, C 0.000 }
gfCNCPoint2[22005] = {X 516.3652, Y 8.5721, Z -3.0000, A 0.000, B 0.000, C 0.000 }
gfCNCPoint2[22006] = {X 516.8418, Y 7.8137, Z -3.0000, A 0.000, B 0.000, C 0.000 }
gfCNCPoint2[22007] = {X 517.4752, Y 7.1803, Z -3.0000, A 0.000, B 0.000, C 0.000 }
gfCNCPoint2[22008] = {X 518.2337, Y 6.7038, Z -3.0000, A 0.000, B 0.000, C 0.000 }
gfCNCPoint2[22009] = {X 519.0791, Y 6.4080, Z -3.0000, A 0.000, B 0.000, C 0.000 }
gfCNCPoint2[22010] = {X 519.9692, Y 6.3077, Z -3.0000, A 0.000, B 0.000, C 0.000 }
gfCNCPoint2[22011] = {X 520.6473, Y 6.3079, Z -3.0000, A 0.000, B 0.000, C 0.000 }
gfCNCPoint2[22012] = {X 521.4443, Y 6.3955, Z -3.0000, A 0.000, B 0.000, C 0.000 }
gfCNCPoint2[22013] = {X 522.2078, Y 6.6403, Z -3.0000, A 0.000, B 0.000, C 0.000 }
gfCNCPoint2[22014] = {X 522.9072, Y 7.0325, Z -3.0000, A 0.000, B 0.000, C 0.000 }
gfCNCPoint2[22015] = {X 523.5142, Y 7.5563, Z -3.0000, A 0.000, B 0.000, C 0.000 }
gfCNCPoint2[22016] = {X 524.0046, Y 8.1907, Z -3.0000, A 0.000, B 0.000, C 0.000 }
gfCNCPoint2[22017] = {X 533.9638, Y 8.1910, Z -3.0000, A 0.000, B 0.000, C 0.000 }
gfCNCPoint2[22018] = {X 533.9640, Y 4.1110, Z -3.0000, A 0.000, B 0.000, C 0.000 }
gfCNCPoint2[22019] = {X 533.9640, Y 4.1110, Z 0.0000, A 0.000, B 0.000, C 0.000 }
gfCNCPoint2[22020] = {X 533.9640, Y 4.1110, Z 11.0000, A 0.000, B 0.000, C 0.000 }
gfCNCPoint2[22021] = {X 419.6136, Y 26.5283, Z 11.0000, A 0.000, B 0.000, C 0.000 }
gfCNCPoint2[22022] = {X 419.6136, Y 26.5283, Z 0.0000, A 0.000, B 0.000, C 0.000 }
gfCNCPoint2[22023] = {X 419.6136, Y 26.5283, Z -3.0000, A 0.000, B 0.000, C 0.000 }
gfCNCPoint2[22024] = {X 416.1502, Y 24.3716, Z -3.0000, A 0.000, B 0.000, C 0.000 }
gfCNCPoint2[22025] = {X 411.5463, Y 31.7649, Z -3.0000, A 0.000, B 0.000, C 0.000 }
gfCNCPoint2[22026] = {X 411.5470, Y 40.8983, Z -3.0000, A 0.000, B 0.000, C 0.000 }
gfCNCPoint2[22027] = {X 412.1851, Y 41.5841, Z -3.0000, A 0.000, B 0.000, C 0.000 }
gfCNCPoint2[22028] = {X 412.6653, Y 42.3884, Z -3.0000, A 0.000, B 0.000, C 0.000 }
gfCNCPoint2[22029] = {X 412.9663, Y 43.2755, Z -3.0000, A 0.000, B 0.000, C 0.000 }
gfCNCPoint2[22030] = {X 413.0747, Y 44.2060, Z -3.0000, A 0.000, B 0.000, C 0.000 }
gfCNCPoint2[22031] = {X 413.0747, Y 45.0002, Z -3.0000, A 0.000, B 0.000, C 0.000 }
gfCNCPoint2[22032] = {X 412.9663, Y 45.9614, Z -3.0000, A 0.000, B 0.000, C 0.000 }
gfCNCPoint2[22033] = {X 412.6468, Y 46.8745, Z -3.0000, A 0.000, B 0.000, C 0.000 }
gfCNCPoint2[22034] = {X 412.1321, Y 47.6935, Z -3.0000, A 0.000, B 0.000, C 0.000 }
gfCNCPoint2[22035] = {X 411.4481, Y 48.3776, Z -3.0000, A 0.000, B 0.000, C 0.000 }
gfCNCPoint2[22036] = {X 410.6290, Y 48.8922, Z -3.0000, A 0.000, B 0.000, C 0.000 }
gfCNCPoint2[22037] = {X 409.7159, Y 49.2117, Z -3.0000, A 0.000, B 0.000, C 0.000 }
gfCNCPoint2[22038] = {X 408.7547, Y 49.3200, Z -3.0000, A 0.000, B 0.000, C 0.000 }
gfCNCPoint2[22039] = {X 402.3112, Y 49.3200, Z -3.0000, A 0.000, B 0.000, C 0.000 }
gfCNCPoint2[22040] = {X 401.3546, Y 49.2127, Z -3.0000, A 0.000, B 0.000, C 0.000 }
gfCNCPoint2[22041] = {X 400.4455, Y 48.8963, Z -3.0000, A 0.000, B 0.000, C 0.000 }
gfCNCPoint2[22042] = {X 399.6290, Y 48.3864, Z -3.0000, A 0.000, B 0.000, C 0.000 }
gfCNCPoint2[22043] = {X 398.9457, Y 47.7084, Z -3.0000, A 0.000, B 0.000, C 0.000 }
gfCNCPoint2[22044] = {X 398.4295, Y 46.8959, Z -3.0000, A 0.000, B 0.000, C 0.000 }
gfCNCPoint2[22045] = {X 398.1060, Y 45.9892, Z -3.0000, A 0.000, B 0.000, C 0.000 }
gfCNCPoint2[22046] = {X 397.9913, Y 45.0335, Z -3.0000, A 0.000, B 0.000, C 0.000 }
gfCNCPoint2[22047] = {X 397.9916, Y 44.1528, Z -3.0000, A 0.000, B 0.000, C 0.000 }
gfCNCPoint2[22048] = {X 398.1015, Y 43.2391, Z -3.0000, A 0.000, B 0.000, C 0.000 }
gfCNCPoint2[22049] = {X 398.4024, Y 42.3694, Z -3.0000, A 0.000, B 0.000, C 0.000 }
gfCNCPoint2[22050] = {X 398.8807, Y 41.5832, Z -3.0000, A 0.000, B 0.000, C 0.000 }
gfCNCPoint2[22051] = {X 399.5147, Y 40.9161, Z -3.0000, A 0.000, B 0.000, C 0.000 }
gfCNCPoint2[22052] = {X 399.4728, Y 31.5991, Z -3.0000, A 0.000, B 0.000, C 0.000 }
gfCNCPoint2[22053] = {X 395.2853, Y 24.3204, Z -3.0000, A 0.000, B 0.000, C 0.000 }
gfCNCPoint2[22054] = {X 393.5914, Y 21.3666, Z -3.0000, A 0.000, B 0.000, C 0.000 }
gfCNCPoint2[22055] = {X 392.6480, Y 19.7615, Z -3.0000, A 0.000, B 0.000, C 0.000 }
gfCNCPoint2[22056] = {X 391.6705, Y 18.1769, Z -3.0000, A 0.000, B 0.000, C 0.000 }
gfCNCPoint2[22057] = {X 391.2080, Y 17.5391, Z -3.0000, A 0.000, B 0.000, C 0.000 }
gfCNCPoint2[22058] = {X 390.6678, Y 16.9656, Z -3.0000, A 0.000, B 0.000, C 0.000 }
gfCNCPoint2[22059] = {X 389.7908, Y 16.4733, Z -3.0000, A 0.000, B 0.000, C 0.000 }
gfCNCPoint2[22060] = {X 389.0514, Y 15.7915, Z -3.0000, A 0.000, B 0.000, C 0.000 }
gfCNCPoint2[22061] = {X 388.4897, Y 14.9573, Z -3.0000, A 0.000, B 0.000, C 0.000 }
gfCNCPoint2[22062] = {X 388.1361, Y 14.0158, Z -3.0000, A 0.000, B 0.000, C 0.000 }
gfCNCPoint2[22063] = {X 388.0098, Y 13.0180, Z -3.0000, A 0.000, B 0.000, C 0.000 }
gfCNCPoint2[22064] = {X 388.0096, Y 12.1868, Z -3.0000, A 0.000, B 0.000, C 0.000 }
gfCNCPoint2[22065] = {X 388.1179, Y 11.2255, Z -3.0000, A 0.000, B 0.000, C 0.000 }
gfCNCPoint2[22066] = {X 388.4374, Y 10.3125, Z -3.0000, A 0.000, B 0.000, C 0.000 }
gfCNCPoint2[22067] = {X 388.9521, Y 9.4933, Z -3.0000, A 0.000, B 0.000, C 0.000 }
gfCNCPoint2[22068] = {X 389.6361, Y 8.8093, Z -3.0000, A 0.000, B 0.000, C 0.000 }
gfCNCPoint2[22069] = {X 390.4552, Y 8.2946, Z -3.0000, A 0.000, B 0.000, C 0.000 }
gfCNCPoint2[22070] = {X 391.3683, Y 7.9751, Z -3.0000, A 0.000, B 0.000, C 0.000 }
gfCNCPoint2[22071] = {X 392.3296, Y 7.8668, Z -3.0000, A 0.000, B 0.000, C 0.000 }
gfCNCPoint2[22072] = {X 399.1118, Y 7.8668, Z -3.0000, A 0.000, B 0.000, C 0.000 }
gfCNCPoint2[22073] = {X 400.0730, Y 7.9751, Z -3.0000, A 0.000, B 0.000, C 0.000 }
gfCNCPoint2[22074] = {X 400.9861, Y 8.2946, Z -3.0000, A 0.000, B 0.000, C 0.000 }
gfCNCPoint2[22075] = {X 401.8052, Y 8.8093, Z -3.0000, A 0.000, B 0.000, C 0.000 }
gfCNCPoint2[22076] = {X 402.4893, Y 9.4933, Z -3.0000, A 0.000, B 0.000, C 0.000 }
gfCNCPoint2[22077] = {X 403.0039, Y 10.3124, Z -3.0000, A 0.000, B 0.000, C 0.000 }
gfCNCPoint2[22078] = {X 403.3234, Y 11.2255, Z -3.0000, A 0.000, B 0.000, C 0.000 }
gfCNCPoint2[22079] = {X 403.4318, Y 12.1868, Z -3.0000, A 0.000, B 0.000, C 0.000 }
gfCNCPoint2[22080] = {X 403.4318, Y 12.9781, Z -3.0000, A 0.000, B 0.000, C 0.000 }
gfCNCPoint2[22081] = {X 403.3293, Y 13.9134, Z -3.0000, A 0.000, B 0.000, C 0.000 }
gfCNCPoint2[22082] = {X 403.0267, Y 14.8043, Z -3.0000, A 0.000, B 0.000, C 0.000 }
gfCNCPoint2[22083] = {X 405.3568, Y 18.8235, Z -3.0000, A 0.000, B 0.000, C 0.000 }
gfCNCPoint2[22084] = {X 407.8736, Y 14.7543, Z -3.0000, A 0.000, B 0.000, C 0.000 }
gfCNCPoint2[22085] = {X 407.5921, Y 13.9046, Z -3.0000, A 0.000, B 0.000, C 0.000 }
gfCNCPoint2[22086] = {X 407.4917, Y 13.0151, Z -3.0000, A 0.000, B 0.000, C 0.000 }
gfCNCPoint2[22087] = {X 407.4915, Y 12.1868, Z -3.0000, A 0.000, B 0.000, C 0.000 }
gfCNCPoint2[22088] = {X 407.5999, Y 11.2255, Z -3.0000, A 0.000, B 0.000, C 0.000 }
gfCNCPoint2[22089] = {X 407.9194, Y 10.3124, Z -3.0000, A 0.000, B 0.000, C 0.000 }
gfCNCPoint2[22090] = {X 408.4340, Y 9.4933, Z -3.0000, A 0.000, B 0.000, C 0.000 }
gfCNCPoint2[22091] = {X 409.1181, Y 8.8093, Z -3.0000, A 0.000, B 0.000, C 0.000 }
gfCNCPoint2[22092] = {X 409.9372, Y 8.2946, Z -3.0000, A 0.000, B 0.000, C 0.000 }
gfCNCPoint2[22093] = {X 410.8502, Y 7.9751, Z -3.0000, A 0.000, B 0.000, C 0.000 }
gfCNCPoint2[22094] = {X 411.8115, Y 7.8668, Z -3.0000, A 0.000, B 0.000, C 0.000 }
gfCNCPoint2[22095] = {X 419.3245, Y 7.8668, Z -3.0000, A 0.000, B 0.000, C 0.000 }
gfCNCPoint2[22096] = {X 420.2858, Y 7.9751, Z -3.0000, A 0.000, B 0.000, C 0.000 }
gfCNCPoint2[22097] = {X 421.1988, Y 8.2946, Z -3.0000, A 0.000, B 0.000, C 0.000 }
gfCNCPoint2[22098] = {X 422.0179, Y 8.8093, Z -3.0000, A 0.000, B 0.000, C 0.000 }
gfCNCPoint2[22099] = {X 422.7020, Y 9.4933, Z -3.0000, A 0.000, B 0.000, C 0.000 }
gfCNCPoint2[22100] = {X 423.2166, Y 10.3124, Z -3.0000, A 0.000, B 0.000, C 0.000 }
gfCNCPoint2[22101] = {X 423.5361, Y 11.2255, Z -3.0000, A 0.000, B 0.000, C 0.000 }
gfCNCPoint2[22102] = {X 423.6445, Y 12.1868, Z -3.0000, A 0.000, B 0.000, C 0.000 }
gfCNCPoint2[22103] = {X 423.6445, Y 12.9804, Z -3.0000, A 0.000, B 0.000, C 0.000 }
gfCNCPoint2[22104] = {X 423.5512, Y 13.8469, Z -3.0000, A 0.000, B 0.000, C 0.000 }
gfCNCPoint2[22105] = {X 423.2884, Y 14.6778, Z -3.0000, A 0.000, B 0.000, C 0.000 }
gfCNCPoint2[22106] = {X 422.8666, Y 15.4404, Z -3.0000, A 0.000, B 0.000, C 0.000 }
gfCNCPoint2[22107] = {X 422.3023, Y 16.1046, Z -3.0000, A 0.000, B 0.000, C 0.000 }
gfCNCPoint2[22108] = {X 421.6179, Y 16.6440, Z -3.0000, A 0.000, B 0.000, C 0.000 }
gfCNCPoint2[22109] = {X 420.8403, Y 17.0375, Z -3.0000, A 0.000, B 0.000, C 0.000 }
gfCNCPoint2[22110] = {X 420.1239, Y 18.0010, Z -3.0000, A 0.000, B 0.000, C 0.000 }
gfCNCPoint2[22111] = {X 419.4756, Y 19.0115, Z -3.0000, A 0.000, B 0.000, C 0.000 }
gfCNCPoint2[22112] = {X 417.9942, Y 21.4103, Z -3.0000, A 0.000, B 0.000, C 0.000 }
gfCNCPoint2[22113] = {X 416.1502, Y 24.3716, Z -3.0000, A 0.000, B 0.000, C 0.000 }
gfCNCPoint2[22114] = {X 419.5457, Y 26.4861, Z -3.0000, A 0.000, B 0.000, C 0.000 }
gfCNCPoint2[22115] = {X 416.0823, Y 24.3294, Z -3.0000, A 0.000, B 0.000, C 0.000 }
gfCNCPoint2[22116] = {X 411.4663, Y 31.7421, Z -3.0000, A 0.000, B 0.000, C 0.000 }
gfCNCPoint2[22117] = {X 411.4670, Y 40.9349, Z -3.0000, A 0.000, B 0.000, C 0.000 }
gfCNCPoint2[22118] = {X 412.1047, Y 41.6104, Z -3.0000, A 0.000, B 0.000, C 0.000 }
gfCNCPoint2[22119] = {X 412.5850, Y 42.4055, Z -3.0000, A 0.000, B 0.000, C 0.000 }
gfCNCPoint2[22120] = {X 412.8862, Y 43.2842, Z -3.0000, A 0.000, B 0.000, C 0.000 }
gfCNCPoint2[22121] = {X 412.9947, Y 44.2068, Z -3.0000, A 0.000, B 0.000, C 0.000 }
gfCNCPoint2[22122] = {X 412.9947, Y 45.0002, Z -3.0000, A 0.000, B 0.000, C 0.000 }
gfCNCPoint2[22123] = {X 412.8883, Y 45.9436, Z -3.0000, A 0.000, B 0.000, C 0.000 }
gfCNCPoint2[22124] = {X 412.5747, Y 46.8398, Z -3.0000, A 0.000, B 0.000, C 0.000 }
gfCNCPoint2[22125] = {X 412.0696, Y 47.6437, Z -3.0000, A 0.000, B 0.000, C 0.000 }
gfCNCPoint2[22126] = {X 411.3982, Y 48.3150, Z -3.0000, A 0.000, B 0.000, C 0.000 }
gfCNCPoint2[22127] = {X 410.5943, Y 48.8201, Z -3.0000, A 0.000, B 0.000, C 0.000 }
gfCNCPoint2[22128] = {X 409.6981, Y 49.1337, Z -3.0000, A 0.000, B 0.000, C 0.000 }
gfCNCPoint2[22129] = {X 408.7547, Y 49.2400, Z -3.0000, A 0.000, B 0.000, C 0.000 }
gfCNCPoint2[22130] = {X 402.3112, Y 49.2400, Z -3.0000, A 0.000, B 0.000, C 0.000 }
gfCNCPoint2[22131] = {X 401.3723, Y 49.1347, Z -3.0000, A 0.000, B 0.000, C 0.000 }
gfCNCPoint2[22132] = {X 400.4800, Y 48.8242, Z -3.0000, A 0.000, B 0.000, C 0.000 }
gfCNCPoint2[22133] = {X 399.6786, Y 48.3237, Z -3.0000, A 0.000, B 0.000, C 0.000 }
gfCNCPoint2[22134] = {X 399.0080, Y 47.6582, Z -3.0000, A 0.000, B 0.000, C 0.000 }
gfCNCPoint2[22135] = {X 398.5013, Y 46.8608, Z -3.0000, A 0.000, B 0.000, C 0.000 }
gfCNCPoint2[22136] = {X 398.1839, Y 45.9709, Z -3.0000, A 0.000, B 0.000, C 0.000 }
gfCNCPoint2[22137] = {X 398.0713, Y 45.0329, Z -3.0000, A 0.000, B 0.000, C 0.000 }
gfCNCPoint2[22138] = {X 398.0716, Y 44.1538, Z -3.0000, A 0.000, B 0.000, C 0.000 }
gfCNCPoint2[22139] = {X 398.1815, Y 43.2480, Z -3.0000, A 0.000, B 0.000, C 0.000 }
gfCNCPoint2[22140] = {X 398.4827, Y 42.3867, Z -3.0000, A 0.000, B 0.000, C 0.000 }
gfCNCPoint2[22141] = {X 398.9612, Y 41.6098, Z -3.0000, A 0.000, B 0.000, C 0.000 }
gfCNCPoint2[22142] = {X 399.5948, Y 40.9532, Z -3.0000, A 0.000, B 0.000, C 0.000 }
gfCNCPoint2[22143] = {X 399.5527, Y 31.5775, Z -3.0000, A 0.000, B 0.000, C 0.000 }
gfCNCPoint2[22144] = {X 395.3547, Y 24.2806, Z -3.0000, A 0.000, B 0.000, C 0.000 }
gfCNCPoint2[22145] = {X 393.6608, Y 21.3268, Z -3.0000, A 0.000, B 0.000, C 0.000 }
gfCNCPoint2[22146] = {X 392.7165, Y 19.7202, Z -3.0000, A 0.000, B 0.000, C 0.000 }
gfCNCPoint2[22147] = {X 391.7382, Y 18.1341, Z -3.0000, A 0.000, B 0.000, C 0.000 }
gfCNCPoint2[22148] = {X 391.2650, Y 17.4825, Z -3.0000, A 0.000, B 0.000, C 0.000 }
gfCNCPoint2[22149] = {X 390.7118, Y 16.8972, Z -3.0000, A 0.000, B 0.000, C 0.000 }
gfCNCPoint2[22150] = {X 389.8471, Y 16.4153, Z -3.0000, A 0.000, B 0.000, C 0.000 }
gfCNCPoint2[22151] = {X 389.1177, Y 15.7459, Z -3.0000, A 0.000, B 0.000, C 0.000 }
gfCNCPoint2[22152] = {X 388.5635, Y 14.9257, Z -3.0000, A 0.000, B 0.000, C 0.000 }
gfCNCPoint2[22153] = {X 388.2145, Y 13.9994, Z -3.0000, A 0.000, B 0.000, C 0.000 }
gfCNCPoint2[22154] = {X 388.0898, Y 13.0173, Z -3.0000, A 0.000, B 0.000, C 0.000 }
gfCNCPoint2[22155] = {X 388.0896, Y 12.1868, Z -3.0000, A 0.000, B 0.000, C 0.000 }
gfCNCPoint2[22156] = {X 388.1959, Y 11.2433, Z -3.0000, A 0.000, B 0.000, C 0.000 }
gfCNCPoint2[22157] = {X 388.5095, Y 10.3472, Z -3.0000, A 0.000, B 0.000, C 0.000 }
gfCNCPoint2[22158] = {X 389.0147, Y 9.5432, Z -3.0000, A 0.000, B 0.000, C 0.000 }
gfCNCPoint2[22159] = {X 389.6860, Y 8.8719, Z -3.0000, A 0.000, B 0.000, C 0.000 }
gfCNCPoint2[22160] = {X 390.4900, Y 8.3667, Z -3.0000, A 0.000, B 0.000, C 0.000 }
gfCNCPoint2[22161] = {X 391.3861, Y 8.0531, Z -3.0000, A 0.000, B 0.000, C 0.000 }
gfCNCPoint2[22162] = {X 392.3296, Y 7.9468, Z -3.0000, A 0.000, B 0.000, C 0.000 }
gfCNCPoint2[22163] = {X 399.1118, Y 7.9468, Z -3.0000, A 0.000, B 0.000, C 0.000 }
gfCNCPoint2[22164] = {X 400.0552, Y 8.0531, Z -3.0000, A 0.000, B 0.000, C 0.000 }
gfCNCPoint2[22165] = {X 400.9514, Y 8.3667, Z -3.0000, A 0.000, B 0.000, C 0.000 }
gfCNCPoint2[22166] = {X 401.7554, Y 8.8718, Z -3.0000, A 0.000, B 0.000, C 0.000 }
gfCNCPoint2[22167] = {X 402.4267, Y 9.5432, Z -3.0000, A 0.000, B 0.000, C 0.000 }
gfCNCPoint2[22168] = {X 402.9319, Y 10.3471, Z -3.0000, A 0.000, B 0.000, C 0.000 }
gfCNCPoint2[22169] = {X 403.2455, Y 11.2433, Z -3.0000, A 0.000, B 0.000, C 0.000 }
gfCNCPoint2[22170] = {X 403.3518, Y 12.1868, Z -3.0000, A 0.000, B 0.000, C 0.000 }
gfCNCPoint2[22171] = {X 403.3518, Y 12.9781, Z -3.0000, A 0.000, B 0.000, C 0.000 }
gfCNCPoint2[22172] = {X 403.2466, Y 13.9164, Z -3.0000, A 0.000, B 0.000, C 0.000 }
gfCNCPoint2[22173] = {X 402.9365, Y 14.8081, Z -3.0000, A 0.000, B 0.000, C 0.000 }
gfCNCPoint2[22174] = {X 405.3546, Y 18.9791, Z -3.0000, A 0.000, B 0.000, C 0.000 }
gfCNCPoint2[22175] = {X 407.9642, Y 14.7599, Z -3.0000, A 0.000, B 0.000, C 0.000 }
gfCNCPoint2[22176] = {X 407.6748, Y 13.9081, Z -3.0000, A 0.000, B 0.000, C 0.000 }
gfCNCPoint2[22177] = {X 407.5717, Y 13.0144, Z -3.0000, A 0.000, B 0.000, C 0.000 }
gfCNCPoint2[22178] = {X 407.5715, Y 12.1868, Z -3.0000, A 0.000, B 0.000, C 0.000 }
gfCNCPoint2[22179] = {X 407.6778, Y 11.2433, Z -3.0000, A 0.000, B 0.000, C 0.000 }
gfCNCPoint2[22180] = {X 407.9914, Y 10.3471, Z -3.0000, A 0.000, B 0.000, C 0.000 }
gfCNCPoint2[22181] = {X 408.4966, Y 9.5432, Z -3.0000, A 0.000, B 0.000, C 0.000 }
gfCNCPoint2[22182] = {X 409.1679, Y 8.8718, Z -3.0000, A 0.000, B 0.000, C 0.000 }
gfCNCPoint2[22183] = {X 409.9719, Y 8.3667, Z -3.0000, A 0.000, B 0.000, C 0.000 }
gfCNCPoint2[22184] = {X 410.8680, Y 8.0531, Z -3.0000, A 0.000, B 0.000, C 0.000 }
gfCNCPoint2[22185] = {X 411.8115, Y 7.9468, Z -3.0000, A 0.000, B 0.000, C 0.000 }
gfCNCPoint2[22186] = {X 419.3245, Y 7.9468, Z -3.0000, A 0.000, B 0.000, C 0.000 }
gfCNCPoint2[22187] = {X 420.2679, Y 8.0531, Z -3.0000, A 0.000, B 0.000, C 0.000 }
gfCNCPoint2[22188] = {X 421.1641, Y 8.3667, Z -3.0000, A 0.000, B 0.000, C 0.000 }
gfCNCPoint2[22189] = {X 421.9681, Y 8.8718, Z -3.0000, A 0.000, B 0.000, C 0.000 }
gfCNCPoint2[22190] = {X 422.6394, Y 9.5432, Z -3.0000, A 0.000, B 0.000, C 0.000 }
gfCNCPoint2[22191] = {X 423.1446, Y 10.3471, Z -3.0000, A 0.000, B 0.000, C 0.000 }
gfCNCPoint2[22192] = {X 423.4582, Y 11.2433, Z -3.0000, A 0.000, B 0.000, C 0.000 }
gfCNCPoint2[22193] = {X 423.5645, Y 12.1868, Z -3.0000, A 0.000, B 0.000, C 0.000 }
gfCNCPoint2[22194] = {X 423.5645, Y 12.9798, Z -3.0000, A 0.000, B 0.000, C 0.000 }
gfCNCPoint2[22195] = {X 423.4721, Y 13.8340, Z -3.0000, A 0.000, B 0.000, C 0.000 }
gfCNCPoint2[22196] = {X 423.2121, Y 14.6529, Z -3.0000, A 0.000, B 0.000, C 0.000 }
gfCNCPoint2[22197] = {X 422.7947, Y 15.4038, Z -3.0000, A 0.000, B 0.000, C 0.000 }
gfCNCPoint2[22198] = {X 422.2365, Y 16.0569, Z -3.0000, A 0.000, B 0.000, C 0.000 }
gfCNCPoint2[22199] = {X 421.5597, Y 16.5862, Z -3.0000, A 0.000, B 0.000, C 0.000 }
gfCNCPoint2[22200] = {X 420.7913, Y 16.9706, Z -3.0000, A 0.000, B 0.000, C 0.000 }
gfCNCPoint2[22201] = {X 420.0645, Y 17.9463, Z -3.0000, A 0.000, B 0.000, C 0.000 }
gfCNCPoint2[22202] = {X 419.4071, Y 18.9701, Z -3.0000, A 0.000, B 0.000, C 0.000 }
gfCNCPoint2[22203] = {X 417.9262, Y 21.3682, Z -3.0000, A 0.000, B 0.000, C 0.000 }
gfCNCPoint2[22204] = {X 416.0823, Y 24.3294, Z -3.0000, A 0.000, B 0.000, C 0.000 }
gfCNCPoint2[22205] = {X 419.4778, Y 26.4438, Z -3.0000, A 0.000, B 0.000, C 0.000 }
gfCNCPoint2[22206] = {X 416.0144, Y 24.2871, Z -3.0000, A 0.000, B 0.000, C 0.000 }
gfCNCPoint2[22207] = {X 411.3863, Y 31.7192, Z -3.0000, A 0.000, B 0.000, C 0.000 }
gfCNCPoint2[22208] = {X 411.3870, Y 40.9720, Z -3.0000, A 0.000, B 0.000, C 0.000 }
gfCNCPoint2[22209] = {X 412.0243, Y 41.6369, Z -3.0000, A 0.000, B 0.000, C 0.000 }
gfCNCPoint2[22210] = {X 412.5047, Y 42.4227, Z -3.0000, A 0.000, B 0.000, C 0.000 }
gfCNCPoint2[22211] = {X 412.8062, Y 43.2930, Z -3.0000, A 0.000, B 0.000, C 0.000 }
gfCNCPoint2[22212] = {X 412.9147, Y 44.2076, Z -3.0000, A 0.000, B 0.000, C 0.000 }
gfCNCPoint2[22213] = {X 412.9147, Y 45.0002, Z -3.0000, A 0.000, B 0.000, C 0.000 }
gfCNCPoint2[22214] = {X 412.8103, Y 45.9258, Z -3.0000, A 0.000, B 0.000, C 0.000 }
gfCNCPoint2[22215] = {X 412.5027, Y 46.8051, Z -3.0000, A 0.000, B 0.000, C 0.000 }
gfCNCPoint2[22216] = {X 412.0070, Y 47.5938, Z -3.0000, A 0.000, B 0.000, C 0.000 }
gfCNCPoint2[22217] = {X 411.3483, Y 48.2525, Z -3.0000, A 0.000, B 0.000, C 0.000 }
gfCNCPoint2[22218] = {X 410.5596, Y 48.7480, Z -3.0000, A 0.000, B 0.000, C 0.000 }
gfCNCPoint2[22219] = {X 409.6803, Y 49.0557, Z -3.0000, A 0.000, B 0.000, C 0.000 }
gfCNCPoint2[22220] = {X 408.7547, Y 49.1600, Z -3.0000, A 0.000, B 0.000, C 0.000 }
gfCNCPoint2[22221] = {X 402.3112, Y 49.1600, Z -3.0000, A 0.000, B 0.000, C 0.000 }
gfCNCPoint2[22222] = {X 401.3900, Y 49.0567, Z -3.0000, A 0.000, B 0.000, C 0.000 }
gfCNCPoint2[22223] = {X 400.5146, Y 48.7520, Z -3.0000, A 0.000, B 0.000, C 0.000 }
gfCNCPoint2[22224] = {X 399.7283, Y 48.2610, Z -3.0000, A 0.000, B 0.000, C 0.000 }
gfCNCPoint2[22225] = {X 399.0703, Y 47.6081, Z -3.0000, A 0.000, B 0.000, C 0.000 }
gfCNCPoint2[22226] = {X 398.5732, Y 46.8257, Z -3.0000, A 0.000, B 0.000, C 0.000 }
gfCNCPoint2[22227] = {X 398.2617, Y 45.9526, Z -3.0000, A 0.000, B 0.000, C 0.000 }
gfCNCPoint2[22228] = {X 398.1513, Y 45.0322, Z -3.0000, A 0.000, B 0.000, C 0.000 }
gfCNCPoint2[22229] = {X 398.1516, Y 44.1549, Z -3.0000, A 0.000, B 0.000, C 0.000 }
gfCNCPoint2[22230] = {X 398.2616, Y 43.2570, Z -3.0000, A 0.000, B 0.000, C 0.000 }
gfCNCPoint2[22231] = {X 398.5630, Y 42.4041, Z -3.0000, A 0.000, B 0.000, C 0.000 }
gfCNCPoint2[22232] = {X 399.0417, Y 41.6366, Z -3.0000, A 0.000, B 0.000, C 0.000 }
gfCNCPoint2[22233] = {X 399.6750, Y 40.9907, Z -3.0000, A 0.000, B 0.000, C 0.000 }
gfCNCPoint2[22234] = {X 399.6327, Y 31.5560, Z -3.0000, A 0.000, B 0.000, C 0.000 }
gfCNCPoint2[22235] = {X 395.4240, Y 24.2408, Z -3.0000, A 0.000, B 0.000, C 0.000 }
gfCNCPoint2[22236] = {X 393.7302, Y 21.2870, Z -3.0000, A 0.000, B 0.000, C 0.000 }
gfCNCPoint2[22237] = {X 392.7851, Y 19.6789, Z -3.0000, A 0.000, B 0.000, C 0.000 }
gfCNCPoint2[22238] = {X 391.8058, Y 18.0914, Z -3.0000, A 0.000, B 0.000, C 0.000 }
gfCNCPoint2[22239] = {X 391.3219, Y 17.4258, Z -3.0000, A 0.000, B 0.000, C 0.000 }
gfCNCPoint2[22240] = {X 390.7556, Y 16.8287, Z -3.0000, A 0.000, B 0.000, C 0.000 }
gfCNCPoint2[22241] = {X 389.9032, Y 16.3571, Z -3.0000, A 0.000, B 0.000, C 0.000 }
gfCNCPoint2[22242] = {X 389.1840, Y 15.7002, Z -3.0000, A 0.000, B 0.000, C 0.000 }
gfCNCPoint2[22243] = {X 388.6372, Y 14.8941, Z -3.0000, A 0.000, B 0.000, C 0.000 }
gfCNCPoint2[22244] = {X 388.2928, Y 13.9829, Z -3.0000, A 0.000, B 0.000, C 0.000 }
gfCNCPoint2[22245] = {X 388.1698, Y 13.0166, Z -3.0000, A 0.000, B 0.000, C 0.000 }
gfCNCPoint2[22246] = {X 388.1696, Y 12.1868, Z -3.0000, A 0.000, B 0.000, C 0.000 }
gfCNCPoint2[22247] = {X 388.2739, Y 11.2611, Z -3.0000, A 0.000, B 0.000, C 0.000 }
gfCNCPoint2[22248] = {X 388.5816, Y 10.3819, Z -3.0000, A 0.000, B 0.000, C 0.000 }
gfCNCPoint2[22249] = {X 389.0772, Y 9.5931, Z -3.0000, A 0.000, B 0.000, C 0.000 }
gfCNCPoint2[22250] = {X 389.7359, Y 8.9344, Z -3.0000, A 0.000, B 0.000, C 0.000 }
gfCNCPoint2[22251] = {X 390.5247, Y 8.4388, Z -3.0000, A 0.000, B 0.000, C 0.000 }
gfCNCPoint2[22252] = {X 391.4039, Y 8.1311, Z -3.0000, A 0.000, B 0.000, C 0.000 }
gfCNCPoint2[22253] = {X 392.3296, Y 8.0268, Z -3.0000, A 0.000, B 0.000, C 0.000 }
gfCNCPoint2[22254] = {X 399.1118, Y 8.0268, Z -3.0000, A 0.000, B 0.000, C 0.000 }
gfCNCPoint2[22255] = {X 400.0374, Y 8.1311, Z -3.0000, A 0.000, B 0.000, C 0.000 }
gfCNCPoint2[22256] = {X 400.9167, Y 8.4388, Z -3.0000, A 0.000, B 0.000, C 0.000 }
gfCNCPoint2[22257] = {X 401.7055, Y 8.9344, Z -3.0000, A 0.000, B 0.000, C 0.000 }
gfCNCPoint2[22258] = {X 402.3642, Y 9.5931, Z -3.0000, A 0.000, B 0.000, C 0.000 }
gfCNCPoint2[22259] = {X 402.8598, Y 10.3819, Z -3.0000, A 0.000, B 0.000, C 0.000 }
gfCNCPoint2[22260] = {X 403.1675, Y 11.2611, Z -3.0000, A 0.000, B 0.000, C 0.000 }
gfCNCPoint2[22261] = {X 403.2718, Y 12.1868, Z -3.0000, A 0.000, B 0.000, C 0.000 }
gfCNCPoint2[22262] = {X 403.2718, Y 12.9781, Z -3.0000, A 0.000, B 0.000, C 0.000 }
gfCNCPoint2[22263] = {X 403.1639, Y 13.9192, Z -3.0000, A 0.000, B 0.000, C 0.000 }
gfCNCPoint2[22264] = {X 402.8459, Y 14.8115, Z -3.0000, A 0.000, B 0.000, C 0.000 }
gfCNCPoint2[22265] = {X 405.3524, Y 19.1348, Z -3.0000, A 0.000, B 0.000, C 0.000 }
gfCNCPoint2[22266] = {X 408.0550, Y 14.7652, Z -3.0000, A 0.000, B 0.000, C 0.000 }
gfCNCPoint2[22267] = {X 407.7576, Y 13.9115, Z -3.0000, A 0.000, B 0.000, C 0.000 }
gfCNCPoint2[22268] = {X 407.6517, Y 13.0137, Z -3.0000, A 0.000, B 0.000, C 0.000 }
gfCNCPoint2[22269] = {X 407.6515, Y 12.1868, Z -3.0000, A 0.000, B 0.000, C 0.000 }
gfCNCPoint2[22270] = {X 407.7558, Y 11.2611, Z -3.0000, A 0.000, B 0.000, C 0.000 }
gfCNCPoint2[22271] = {X 408.0635, Y 10.3819, Z -3.0000, A 0.000, B 0.000, C 0.000 }
gfCNCPoint2[22272] = {X 408.5591, Y 9.5931, Z -3.0000, A 0.000, B 0.000, C 0.000 }
gfCNCPoint2[22273] = {X 409.2178, Y 8.9344, Z -3.0000, A 0.000, B 0.000, C 0.000 }
gfCNCPoint2[22274] = {X 410.0066, Y 8.4388, Z -3.0000, A 0.000, B 0.000, C 0.000 }
gfCNCPoint2[22275] = {X 410.8859, Y 8.1311, Z -3.0000, A 0.000, B 0.000, C 0.000 }
gfCNCPoint2[22276] = {X 411.8115, Y 8.0268, Z -3.0000, A 0.000, B 0.000, C 0.000 }
gfCNCPoint2[22277] = {X 419.3245, Y 8.0268, Z -3.0000, A 0.000, B 0.000, C 0.000 }
gfCNCPoint2[22278] = {X 420.2501, Y 8.1311, Z -3.0000, A 0.000, B 0.000, C 0.000 }
gfCNCPoint2[22279] = {X 421.1294, Y 8.4388, Z -3.0000, A 0.000, B 0.000, C 0.000 }
gfCNCPoint2[22280] = {X 421.9182, Y 8.9344, Z -3.0000, A 0.000, B 0.000, C 0.000 }
gfCNCPoint2[22281] = {X 422.5769, Y 9.5931, Z -3.0000, A 0.000, B 0.000, C 0.000 }
gfCNCPoint2[22282] = {X 423.0725, Y 10.3819, Z -3.0000, A 0.000, B 0.000, C 0.000 }
gfCNCPoint2[22283] = {X 423.3802, Y 11.2611, Z -3.0000, A 0.000, B 0.000, C 0.000 }
gfCNCPoint2[22284] = {X 423.4845, Y 12.1868, Z -3.0000, A 0.000, B 0.000, C 0.000 }
gfCNCPoint2[22285] = {X 423.4845, Y 12.9792, Z -3.0000, A 0.000, B 0.000, C 0.000 }
gfCNCPoint2[22286] = {X 423.3931, Y 13.8210, Z -3.0000, A 0.000, B 0.000, C 0.000 }
gfCNCPoint2[22287] = {X 423.1358, Y 14.6278, Z -3.0000, A 0.000, B 0.000, C 0.000 }
gfCNCPoint2[22288] = {X 422.7228, Y 15.3670, Z -3.0000, A 0.000, B 0.000, C 0.000 }
gfCNCPoint2[22289] = {X 422.1707, Y 16.0091, Z -3.0000, A 0.000, B 0.000, C 0.000 }
gfCNCPoint2[22290] = {X 421.5017, Y 16.5282, Z -3.0000, A 0.000, B 0.000, C 0.000 }
gfCNCPoint2[22291] = {X 420.7426, Y 16.9035, Z -3.0000, A 0.000, B 0.000, C 0.000 }
gfCNCPoint2[22292] = {X 420.0052, Y 17.8915, Z -3.0000, A 0.000, B 0.000, C 0.000 }
gfCNCPoint2[22293] = {X 419.3387, Y 18.9286, Z -3.0000, A 0.000, B 0.000, C 0.000 }
gfCNCPoint2[22294] = {X 417.8583, Y 21.3260, Z -3.0000, A 0.000, B 0.000, C 0.000 }
gfCNCPoint2[22295] = {X 416.0144, Y 24.2871, Z -3.0000, A 0.000, B 0.000, C 0.000 }
gfCNCPoint2[22296] = {X 419.4099, Y 26.4015, Z -3.0000, A 0.000, B 0.000, C 0.000 }
gfCNCPoint2[22297] = {X 415.9465, Y 24.2448, Z -3.0000, A 0.000, B 0.000, C 0.000 }
gfCNCPoint2[22298] = {X 411.3063, Y 31.6963, Z -3.0000, A 0.000, B 0.000, C 0.000 }
gfCNCPoint2[22299] = {X 411.3070, Y 41.0094, Z -3.0000, A 0.000, B 0.000, C 0.000 }
gfCNCPoint2[22300] = {X 411.9438, Y 41.6637, Z -3.0000, A 0.000, B 0.000, C 0.000 }
gfCNCPoint2[22301] = {X 412.4244, Y 42.4401, Z -3.0000, A 0.000, B 0.000, C 0.000 }
gfCNCPoint2[22302] = {X 412.7261, Y 43.3019, Z -3.0000, A 0.000, B 0.000, C 0.000 }
gfCNCPoint2[22303] = {X 412.8347, Y 44.2085, Z -3.0000, A 0.000, B 0.000, C 0.000 }
gfCNCPoint2[22304] = {X 412.8347, Y 45.0002, Z -3.0000, A 0.000, B 0.000, C 0.000 }
gfCNCPoint2[22305] = {X 412.7324, Y 45.9080, Z -3.0000, A 0.000, B 0.000, C 0.000 }
gfCNCPoint2[22306] = {X 412.4306, Y 46.7703, Z -3.0000, A 0.000, B 0.000, C 0.000 }
gfCNCPoint2[22307] = {X 411.9445, Y 47.5439, Z -3.0000, A 0.000, B 0.000, C 0.000 }
gfCNCPoint2[22308] = {X 411.2985, Y 48.1899, Z -3.0000, A 0.000, B 0.000, C 0.000 }
gfCNCPoint2[22309] = {X 410.5249, Y 48.6760, Z -3.0000, A 0.000, B 0.000, C 0.000 }
gfCNCPoint2[22310] = {X 409.6625, Y 48.9777, Z -3.0000, A 0.000, B 0.000, C 0.000 }
gfCNCPoint2[22311] = {X 408.7547, Y 49.0800, Z -3.0000, A 0.000, B 0.000, C 0.000 }
gfCNCPoint2[22312] = {X 402.3112, Y 49.0800, Z -3.0000, A 0.000, B 0.000, C 0.000 }
gfCNCPoint2[22313] = {X 401.4077, Y 48.9787, Z -3.0000, A 0.000, B 0.000, C 0.000 }
gfCNCPoint2[22314] = {X 400.5491, Y 48.6799, Z -3.0000, A 0.000, B 0.000, C 0.000 }
gfCNCPoint2[22315] = {X 399.7780, Y 48.1983, Z -3.0000, A 0.000, B 0.000, C 0.000 }
gfCNCPoint2[22316] = {X 399.1326, Y 47.5579, Z -3.0000, A 0.000, B 0.000, C 0.000 }
gfCNCPoint2[22317] = {X 398.6451, Y 46.7906, Z -3.0000, A 0.000, B 0.000, C 0.000 }
gfCNCPoint2[22318] = {X 398.3396, Y 45.9343, Z -3.0000, A 0.000, B 0.000, C 0.000 }
gfCNCPoint2[22319] = {X 398.2313, Y 45.0316, Z -3.0000, A 0.000, B 0.000, C 0.000 }
gfCNCPoint2[22320] = {X 398.2316, Y 44.1559, Z -3.0000, A 0.000, B 0.000, C 0.000 }
gfCNCPoint2[22321] = {X 398.3416, Y 43.2661, Z -3.0000, A 0.000, B 0.000, C 0.000 }
gfCNCPoint2[22322] = {X 398.6434, Y 42.4218, Z -3.0000, A 0.000, B 0.000, C 0.000 }
gfCNCPoint2[22323] = {X 399.1223, Y 41.6638, Z -3.0000, A 0.000, B 0.000, C 0.000 }
gfCNCPoint2[22324] = {X 399.7552, Y 41.0287, Z -3.0000, A 0.000, B 0.000, C 0.000 }
gfCNCPoint2[22325] = {X 399.7126, Y 31.5345, Z -3.0000, A 0.000, B 0.000, C 0.000 }
gfCNCPoint2[22326] = {X 395.4934, Y 24.2009, Z -3.0000, A 0.000, B 0.000, C 0.000 }
gfCNCPoint2[22327] = {X 393.7996, Y 21.2472, Z -3.0000, A 0.000, B 0.000, C 0.000 }
gfCNCPoint2[22328] = {X 392.8536, Y 19.6377, Z -3.0000, A 0.000, B 0.000, C 0.000 }
gfCNCPoint2[22329] = {X 391.8734, Y 18.0487, Z -3.0000, A 0.000, B 0.000, C 0.000 }
gfCNCPoint2[22330] = {X 391.3787, Y 17.3690, Z -3.0000, A 0.000, B 0.000, C 0.000 }
gfCNCPoint2[22331] = {X 390.7992, Y 16.7601, Z -3.0000, A 0.000, B 0.000, C 0.000 }
gfCNCPoint2[22332] = {X 389.9593, Y 16.2988, Z -3.0000, A 0.000, B 0.000, C 0.000 }
gfCNCPoint2[22333] = {X 389.2501, Y 15.6544, Z -3.0000, A 0.000, B 0.000, C 0.000 }
gfCNCPoint2[22334] = {X 388.7108, Y 14.8623, Z -3.0000, A 0.000, B 0.000, C 0.000 }
gfCNCPoint2[22335] = {X 388.3711, Y 13.9663, Z -3.0000, A 0.000, B 0.000, C 0.000 }
gfCNCPoint2[22336] = {X 388.2498, Y 13.0158, Z -3.0000, A 0.000, B 0.000, C 0.000 }
gfCNCPoint2[22337] = {X 388.2496, Y 12.1868, Z -3.0000, A 0.000, B 0.000, C 0.000 }
gfCNCPoint2[22338] = {X 388.3519, Y 11.2789, Z -3.0000, A 0.000, B 0.000, C 0.000 }
gfCNCPoint2[22339] = {X 388.6537, Y 10.4166, Z -3.0000, A 0.000, B 0.000, C 0.000 }
gfCNCPoint2[22340] = {X 389.1398, Y 9.6430, Z -3.0000, A 0.000, B 0.000, C 0.000 }
gfCNCPoint2[22341] = {X 389.7858, Y 8.9969, Z -3.0000, A 0.000, B 0.000, C 0.000 }
gfCNCPoint2[22342] = {X 390.5594, Y 8.5109, Z -3.0000, A 0.000, B 0.000, C 0.000 }
gfCNCPoint2[22343] = {X 391.4217, Y 8.2091, Z -3.0000, A 0.000, B 0.000, C 0.000 }
gfCNCPoint2[22344] = {X 392.3296, Y 8.1068, Z -3.0000, A 0.000, B 0.000, C 0.000 }
gfCNCPoint2[22345] = {X 399.1118, Y 8.1068, Z -3.0000, A 0.000, B 0.000, C 0.000 }
gfCNCPoint2[22346] = {X 400.0196, Y 8.2091, Z -3.0000, A 0.000, B 0.000, C 0.000 }
gfCNCPoint2[22347] = {X 400.8820, Y 8.5109, Z -3.0000, A 0.000, B 0.000, C 0.000 }
gfCNCPoint2[22348] = {X 401.6556, Y 8.9969, Z -3.0000, A 0.000, B 0.000, C 0.000 }
gfCNCPoint2[22349] = {X 402.3016, Y 9.6430, Z -3.0000, A 0.000, B 0.000, C 0.000 }
gfCNCPoint2[22350] = {X 402.7877, Y 10.4166, Z -3.0000, A 0.000, B 0.000, C 0.000 }
gfCNCPoint2[22351] = {X 403.0895, Y 11.2789, Z -3.0000, A 0.000, B 0.000, C 0.000 }
gfCNCPoint2[22352] = {X 403.1918, Y 12.1868, Z -3.0000, A 0.000, B 0.000, C 0.000 }
gfCNCPoint2[22353] = {X 403.1918, Y 12.9781, Z -3.0000, A 0.000, B 0.000, C 0.000 }
gfCNCPoint2[22354] = {X 403.0811, Y 13.9219, Z -3.0000, A 0.000, B 0.000, C 0.000 }
gfCNCPoint2[22355] = {X 402.7551, Y 14.8144, Z -3.0000, A 0.000, B 0.000, C 0.000 }
gfCNCPoint2[22356] = {X 405.3502, Y 19.2905, Z -3.0000, A 0.000, B 0.000, C 0.000 }
gfCNCPoint2[22357] = {X 408.1461, Y 14.7699, Z -3.0000, A 0.000, B 0.000, C 0.000 }
gfCNCPoint2[22358] = {X 408.1094, Y 14.6929, Z -3.0000, A 0.000, B 0.000, C 0.000 }
gfCNCPoint2[22359] = {X 408.0744, Y 14.6150, Z -3.0000, A 0.000, B 0.000, C 0.000 }
gfCNCPoint2[22360] = {X 407.8218, Y 13.8314, Z -3.0000, A 0.000, B 0.000, C 0.000 }
gfCNCPoint2[22361] = {X 407.7317, Y 13.0131, Z -3.0000, A 0.000, B 0.000, C 0.000 }
gfCNCPoint2[22362] = {X 407.7315, Y 12.1868, Z -3.0000, A 0.000, B 0.000, C 0.000 }
gfCNCPoint2[22363] = {X 407.8338, Y 11.2789, Z -3.0000, A 0.000, B 0.000, C 0.000 }
gfCNCPoint2[22364] = {X 408.1356, Y 10.4166, Z -3.0000, A 0.000, B 0.000, C 0.000 }
gfCNCPoint2[22365] = {X 408.6217, Y 9.6430, Z -3.0000, A 0.000, B 0.000, C 0.000 }
gfCNCPoint2[22366] = {X 409.2677, Y 8.9969, Z -3.0000, A 0.000, B 0.000, C 0.000 }
gfCNCPoint2[22367] = {X 410.0413, Y 8.5109, Z -3.0000, A 0.000, B 0.000, C 0.000 }
gfCNCPoint2[22368] = {X 410.9037, Y 8.2091, Z -3.0000, A 0.000, B 0.000, C 0.000 }
gfCNCPoint2[22369] = {X 411.8115, Y 8.1068, Z -3.0000, A 0.000, B 0.000, C 0.000 }
gfCNCPoint2[22370] = {X 419.3245, Y 8.1068, Z -3.0000, A 0.000, B 0.000, C 0.000 }
gfCNCPoint2[22371] = {X 420.2323, Y 8.2091, Z -3.0000, A 0.000, B 0.000, C 0.000 }
gfCNCPoint2[22372] = {X 421.0947, Y 8.5109, Z -3.0000, A 0.000, B 0.000, C 0.000 }
gfCNCPoint2[22373] = {X 421.8683, Y 8.9969, Z -3.0000, A 0.000, B 0.000, C 0.000 }
gfCNCPoint2[22374] = {X 422.5143, Y 9.6430, Z -3.0000, A 0.000, B 0.000, C 0.000 }
gfCNCPoint2[22375] = {X 423.0004, Y 10.4166, Z -3.0000, A 0.000, B 0.000, C 0.000 }
gfCNCPoint2[22376] = {X 423.3022, Y 11.2789, Z -3.0000, A 0.000, B 0.000, C 0.000 }
gfCNCPoint2[22377] = {X 423.4045, Y 12.1868, Z -3.0000, A 0.000, B 0.000, C 0.000 }
gfCNCPoint2[22378] = {X 423.4045, Y 12.9786, Z -3.0000, A 0.000, B 0.000, C 0.000 }
gfCNCPoint2[22379] = {X 423.3141, Y 13.8080, Z -3.0000, A 0.000, B 0.000, C 0.000 }
gfCNCPoint2[22380] = {X 423.0595, Y 14.6026, Z -3.0000, A 0.000, B 0.000, C 0.000 }
gfCNCPoint2[22381] = {X 422.6509, Y 15.3302, Z -3.0000, A 0.000, B 0.000, C 0.000 }
gfCNCPoint2[22382] = {X 422.1050, Y 15.9611, Z -3.0000, A 0.000, B 0.000, C 0.000 }
gfCNCPoint2[22383] = {X 421.4438, Y 16.4700, Z -3.0000, A 0.000, B 0.000, C 0.000 }
gfCNCPoint2[22384] = {X 420.6940, Y 16.8362, Z -3.0000, A 0.000, B 0.000, C 0.000 }
gfCNCPoint2[22385] = {X 419.9459, Y 17.8365, Z -3.0000, A 0.000, B 0.000, C 0.000 }
gfCNCPoint2[22386] = {X 419.2703, Y 18.8871, Z -3.0000, A 0.000, B 0.000, C 0.000 }
gfCNCPoint2[22387] = {X 417.7903, Y 21.2839, Z -3.0000, A 0.000, B 0.000, C 0.000 }
gfCNCPoint2[22388] = {X 415.9465, Y 24.2448, Z -3.0000, A 0.000, B 0.000, C 0.000 }
gfCNCPoint2[22389] = {X 419.3419, Y 26.3592, Z -3.0000, A 0.000, B 0.000, C 0.000 }
gfCNCPoint2[22390] = {X 415.8786, Y 24.2025, Z -3.0000, A 0.000, B 0.000, C 0.000 }
gfCNCPoint2[22391] = {X 411.2263, Y 31.6735, Z -3.0000, A 0.000, B 0.000, C 0.000 }
gfCNCPoint2[22392] = {X 411.2270, Y 41.0474, Z -3.0000, A 0.000, B 0.000, C 0.000 }
gfCNCPoint2[22393] = {X 411.8633, Y 41.6908, Z -3.0000, A 0.000, B 0.000, C 0.000 }
gfCNCPoint2[22394] = {X 412.3440, Y 42.4575, Z -3.0000, A 0.000, B 0.000, C 0.000 }
gfCNCPoint2[22395] = {X 412.6460, Y 43.3105, Z -3.0000, A 0.000, B 0.000, C 0.000 }
gfCNCPoint2[22396] = {X 412.7547, Y 44.2089, Z -3.0000, A 0.000, B 0.000, C 0.000 }
gfCNCPoint2[22397] = {X 412.7545, Y 45.0384, Z -3.0000, A 0.000, B 0.000, C 0.000 }
gfCNCPoint2[22398] = {X 412.6469, Y 45.9222, Z -3.0000, A 0.000, B 0.000, C 0.000 }
gfCNCPoint2[22399] = {X 412.3466, Y 46.7602, Z -3.0000, A 0.000, B 0.000, C 0.000 }
gfCNCPoint2[22400] = {X 411.8683, Y 47.5111, Z -3.0000, A 0.000, B 0.000, C 0.000 }
gfCNCPoint2[22401] = {X 411.2357, Y 48.1376, Z -3.0000, A 0.000, B 0.000, C 0.000 }
gfCNCPoint2[22402] = {X 410.4803, Y 48.6086, Z -3.0000, A 0.000, B 0.000, C 0.000 }
gfCNCPoint2[22403] = {X 409.6394, Y 48.9009, Z -3.0000, A 0.000, B 0.000, C 0.000 }
gfCNCPoint2[22404] = {X 408.7547, Y 49.0000, Z -3.0000, A 0.000, B 0.000, C 0.000 }
gfCNCPoint2[22405] = {X 402.3112, Y 49.0000, Z -3.0000, A 0.000, B 0.000, C 0.000 }
gfCNCPoint2[22406] = {X 401.4211, Y 48.8997, Z -3.0000, A 0.000, B 0.000, C 0.000 }
gfCNCPoint2[22407] = {X 400.5757, Y 48.6039, Z -3.0000, A 0.000, B 0.000, C 0.000 }
gfCNCPoint2[22408] = {X 399.8172, Y 48.1273, Z -3.0000, A 0.000, B 0.000, C 0.000 }
gfCNCPoint2[22409] = {X 399.1839, Y 47.4939, Z -3.0000, A 0.000, B 0.000, C 0.000 }
gfCNCPoint2[22410] = {X 398.7073, Y 46.7355, Z -3.0000, A 0.000, B 0.000, C 0.000 }
gfCNCPoint2[22411] = {X 398.4115, Y 45.8900, Z -3.0000, A 0.000, B 0.000, C 0.000 }
gfCNCPoint2[22412] = {X 398.3112, Y 45.0000, Z -3.0000, A 0.000, B 0.000, C 0.000 }
gfCNCPoint2[22413] = {X 398.3115, Y 44.1569, Z -3.0000, A 0.000, B 0.000, C 0.000 }
gfCNCPoint2[22414] = {X 398.4217, Y 43.2753, Z -3.0000, A 0.000, B 0.000, C 0.000 }
gfCNCPoint2[22415] = {X 398.7237, Y 42.4397, Z -3.0000, A 0.000, B 0.000, C 0.000 }
gfCNCPoint2[22416] = {X 399.2028, Y 41.6913, Z -3.0000, A 0.000, B 0.000, C 0.000 }
gfCNCPoint2[22417] = {X 399.8352, Y 41.0672, Z -3.0000, A 0.000, B 0.000, C 0.000 }
gfCNCPoint2[22418] = {X 399.8380, Y 31.5920, Z -3.0000, A 0.000, B 0.000, C 0.000 }
gfCNCPoint2[22419] = {X 395.5628, Y 24.1611, Z -3.0000, A 0.000, B 0.000, C 0.000 }
gfCNCPoint2[22420] = {X 393.8690, Y 21.2074, Z -3.0000, A 0.000, B 0.000, C 0.000 }
gfCNCPoint2[22421] = {X 392.9221, Y 19.5964, Z -3.0000, A 0.000, B 0.000, C 0.000 }
gfCNCPoint2[22422] = {X 391.9411, Y 18.0060, Z -3.0000, A 0.000, B 0.000, C 0.000 }
gfCNCPoint2[22423] = {X 391.4355, Y 17.3122, Z -3.0000, A 0.000, B 0.000, C 0.000 }
gfCNCPoint2[22424] = {X 390.8426, Y 16.6913, Z -3.0000, A 0.000, B 0.000, C 0.000 }
gfCNCPoint2[22425] = {X 390.0091, Y 16.2361, Z -3.0000, A 0.000, B 0.000, C 0.000 }
gfCNCPoint2[22426] = {X 389.3064, Y 15.5972, Z -3.0000, A 0.000, B 0.000, C 0.000 }
gfCNCPoint2[22427] = {X 388.7742, Y 14.8107, Z -3.0000, A 0.000, B 0.000, C 0.000 }
gfCNCPoint2[22428] = {X 388.4423, Y 13.9209, Z -3.0000, A 0.000, B 0.000, C 0.000 }
gfCNCPoint2[22429] = {X 388.3296, Y 12.9779, Z -3.0000, A 0.000, B 0.000, C 0.000 }
gfCNCPoint2[22430] = {X 388.3296, Y 12.1868, Z -3.0000, A 0.000, B 0.000, C 0.000 }
gfCNCPoint2[22431] = {X 388.4299, Y 11.2967, Z -3.0000, A 0.000, B 0.000, C 0.000 }
gfCNCPoint2[22432] = {X 388.7258, Y 10.4513, Z -3.0000, A 0.000, B 0.000, C 0.000 }
gfCNCPoint2[22433] = {X 389.2023, Y 9.6929, Z -3.0000, A 0.000, B 0.000, C 0.000 }
gfCNCPoint2[22434] = {X 389.8357, Y 9.0595, Z -3.0000, A 0.000, B 0.000, C 0.000 }
gfCNCPoint2[22435] = {X 390.5941, Y 8.5829, Z -3.0000, A 0.000, B 0.000, C 0.000 }
gfCNCPoint2[22436] = {X 391.4395, Y 8.2871, Z -3.0000, A 0.000, B 0.000, C 0.000 }
gfCNCPoint2[22437] = {X 392.3296, Y 8.1868, Z -3.0000, A 0.000, B 0.000, C 0.000 }
gfCNCPoint2[22438] = {X 399.1118, Y 8.1868, Z -3.0000, A 0.000, B 0.000, C 0.000 }
gfCNCPoint2[22439] = {X 400.0018, Y 8.2871, Z -3.0000, A 0.000, B 0.000, C 0.000 }
gfCNCPoint2[22440] = {X 400.8473, Y 8.5829, Z -3.0000, A 0.000, B 0.000, C 0.000 }
gfCNCPoint2[22441] = {X 401.6057, Y 9.0595, Z -3.0000, A 0.000, B 0.000, C 0.000 }
gfCNCPoint2[22442] = {X 402.2391, Y 9.6929, Z -3.0000, A 0.000, B 0.000, C 0.000 }
gfCNCPoint2[22443] = {X 402.7156, Y 10.4513, Z -3.0000, A 0.000, B 0.000, C 0.000 }
gfCNCPoint2[22444] = {X 403.0115, Y 11.2967, Z -3.0000, A 0.000, B 0.000, C 0.000 }
gfCNCPoint2[22445] = {X 403.1118, Y 12.1868, Z -3.0000, A 0.000, B 0.000, C 0.000 }
gfCNCPoint2[22446] = {X 403.1115, Y 13.0192, Z -3.0000, A 0.000, B 0.000, C 0.000 }
gfCNCPoint2[22447] = {X 402.9933, Y 13.9442, Z -3.0000, A 0.000, B 0.000, C 0.000 }
gfCNCPoint2[22448] = {X 402.6641, Y 14.8167, Z -3.0000, A 0.000, B 0.000, C 0.000 }
gfCNCPoint2[22449] = {X 405.2576, Y 19.3199, Z -3.0000, A 0.000, B 0.000, C 0.000 }
gfCNCPoint2[22450] = {X 405.3715, Y 19.4083, Z -3.0000, A 0.000, B 0.000, C 0.000 }
gfCNCPoint2[22451] = {X 408.1953, Y 14.8342, Z -3.0000, A 0.000, B 0.000, C 0.000 }
gfCNCPoint2[22452] = {X 408.2428, Y 14.7847, Z -3.0000, A 0.000, B 0.000, C 0.000 }
gfCNCPoint2[22453] = {X 408.1938, Y 14.6845, Z -3.0000, A 0.000, B 0.000, C 0.000 }
gfCNCPoint2[22454] = {X 408.1476, Y 14.5829, Z -3.0000, A 0.000, B 0.000, C 0.000 }
gfCNCPoint2[22455] = {X 407.8965, Y 13.7978, Z -3.0000, A 0.000, B 0.000, C 0.000 }
gfCNCPoint2[22456] = {X 407.8115, Y 12.9779, Z -3.0000, A 0.000, B 0.000, C 0.000 }
gfCNCPoint2[22457] = {X 407.8115, Y 12.1868, Z -3.0000, A 0.000, B 0.000, C 0.000 }
gfCNCPoint2[22458] = {X 407.9118, Y 11.2967, Z -3.0000, A 0.000, B 0.000, C 0.000 }
gfCNCPoint2[22459] = {X 408.2077, Y 10.4513, Z -3.0000, A 0.000, B 0.000, C 0.000 }
gfCNCPoint2[22460] = {X 408.6842, Y 9.6929, Z -3.0000, A 0.000, B 0.000, C 0.000 }
gfCNCPoint2[22461] = {X 409.3176, Y 9.0595, Z -3.0000, A 0.000, B 0.000, C 0.000 }
gfCNCPoint2[22462] = {X 410.0760, Y 8.5829, Z -3.0000, A 0.000, B 0.000, C 0.000 }
gfCNCPoint2[22463] = {X 410.9215, Y 8.2871, Z -3.0000, A 0.000, B 0.000, C 0.000 }
gfCNCPoint2[22464] = {X 411.8115, Y 8.1868, Z -3.0000, A 0.000, B 0.000, C 0.000 }
gfCNCPoint2[22465] = {X 419.3245, Y 8.1868, Z -3.0000, A 0.000, B 0.000, C 0.000 }
gfCNCPoint2[22466] = {X 420.2145, Y 8.2871, Z -3.0000, A 0.000, B 0.000, C 0.000 }
gfCNCPoint2[22467] = {X 421.0600, Y 8.5829, Z -3.0000, A 0.000, B 0.000, C 0.000 }
gfCNCPoint2[22468] = {X 421.8184, Y 9.0595, Z -3.0000, A 0.000, B 0.000, C 0.000 }
gfCNCPoint2[22469] = {X 422.4518, Y 9.6929, Z -3.0000, A 0.000, B 0.000, C 0.000 }
gfCNCPoint2[22470] = {X 422.9283, Y 10.4513, Z -3.0000, A 0.000, B 0.000, C 0.000 }
gfCNCPoint2[22471] = {X 423.2242, Y 11.2967, Z -3.0000, A 0.000, B 0.000, C 0.000 }
gfCNCPoint2[22472] = {X 423.3245, Y 12.1868, Z -3.0000, A 0.000, B 0.000, C 0.000 }
gfCNCPoint2[22473] = {X 423.3245, Y 12.9780, Z -3.0000, A 0.000, B 0.000, C 0.000 }
gfCNCPoint2[22474] = {X 423.1975, Y 13.9553, Z -3.0000, A 0.000, B 0.000, C 0.000 }
gfCNCPoint2[22475] = {X 422.8391, Y 14.8734, Z -3.0000, A 0.000, B 0.000, C 0.000 }
gfCNCPoint2[22476] = {X 422.2703, Y 15.6783, Z -3.0000, A 0.000, B 0.000, C 0.000 }
gfCNCPoint2[22477] = {X 421.5245, Y 16.3227, Z -3.0000, A 0.000, B 0.000, C 0.000 }
gfCNCPoint2[22478] = {X 420.6457, Y 16.7687, Z -3.0000, A 0.000, B 0.000, C 0.000 }
gfCNCPoint2[22479] = {X 419.8867, Y 17.7815, Z -3.0000, A 0.000, B 0.000, C 0.000 }
gfCNCPoint2[22480] = {X 419.2019, Y 18.8457, Z -3.0000, A 0.000, B 0.000, C 0.000 }
gfCNCPoint2[22481] = {X 417.7223, Y 21.2417, Z -3.0000, A 0.000, B 0.000, C 0.000 }
gfCNCPoint2[22482] = {X 415.8786, Y 24.2025, Z -3.0000, A 0.000, B 0.000, C 0.000 }
gfCNCPoint2[22483] = {X 419.3419, Y 26.3592, Z -3.0000, A 0.000, B 0.000, C 0.000 }
gfCNCPoint2[22484] = {X 419.3419, Y 26.3592, Z 0.0000, A 0.000, B 0.000, C 0.000 }
gfCNCPoint2[22485] = {X 419.3419, Y 26.3592, Z 11.0000, A 0.000, B 0.000, C 0.000 }
gfCNCPoint2[22486] = {X 352.3300, Y -3.5329, Z 11.0000, A 0.000, B 0.000, C 0.000 }
gfCNCPoint2[22487] = {X 352.3300, Y -3.5329, Z 0.0000, A 0.000, B 0.000, C 0.000 }
gfCNCPoint2[22488] = {X 352.3300, Y -3.5329, Z -3.0000, A 0.000, B 0.000, C 0.000 }
gfCNCPoint2[22489] = {X 351.5859, Y 0.4787, Z -3.0000, A 0.000, B 0.000, C 0.000 }
gfCNCPoint2[22490] = {X 351.8692, Y 0.5312, Z -3.0000, A 0.000, B 0.000, C 0.000 }
gfCNCPoint2[22491] = {X 353.8039, Y 1.0172, Z -3.0000, A 0.000, B 0.000, C 0.000 }
gfCNCPoint2[22492] = {X 355.6838, Y 1.6844, Z -3.0000, A 0.000, B 0.000, C 0.000 }
gfCNCPoint2[22493] = {X 357.4921, Y 2.5267, Z -3.0000, A 0.000, B 0.000, C 0.000 }
gfCNCPoint2[22494] = {X 359.2124, Y 3.5366, Z -3.0000, A 0.000, B 0.000, C 0.000 }
gfCNCPoint2[22495] = {X 360.8292, Y 4.7050, Z -3.0000, A 0.000, B 0.000, C 0.000 }
gfCNCPoint2[22496] = {X 362.3280, Y 6.0214, Z -3.0000, A 0.000, B 0.000, C 0.000 }
gfCNCPoint2[22497] = {X 363.6953, Y 7.4739, Z -3.0000, A 0.000, B 0.000, C 0.000 }
gfCNCPoint2[22498] = {X 365.1625, Y 9.3674, Z -3.0000, A 0.000, B 0.000, C 0.000 }
gfCNCPoint2[22499] = {X 366.4395, Y 11.3940, Z -3.0000, A 0.000, B 0.000, C 0.000 }
gfCNCPoint2[22500] = {X 367.5144, Y 13.5347, Z -3.0000, A 0.000, B 0.000, C 0.000 }
gfCNCPoint2[22501] = {X 368.3771, Y 15.7693, Z -3.0000, A 0.000, B 0.000, C 0.000 }
gfCNCPoint2[22502] = {X 369.0194, Y 18.0770, Z -3.0000, A 0.000, B 0.000, C 0.000 }
gfCNCPoint2[22503] = {X 369.5005, Y 20.7116, Z -3.0000, A 0.000, B 0.000, C 0.000 }
gfCNCPoint2[22504] = {X 369.7570, Y 23.3775, Z -3.0000, A 0.000, B 0.000, C 0.000 }
gfCNCPoint2[22505] = {X 369.7870, Y 26.0555, Z -3.0000, A 0.000, B 0.000, C 0.000 }
gfCNCPoint2[22506] = {X 369.5903, Y 28.7264, Z -3.0000, A 0.000, B 0.000, C 0.000 }
gfCNCPoint2[22507] = {X 369.1683, Y 31.3712, Z -3.0000, A 0.000, B 0.000, C 0.000 }
gfCNCPoint2[22508] = {X 368.6444, Y 33.4757, Z -3.0000, A 0.000, B 0.000, C 0.000 }
gfCNCPoint2[22509] = {X 367.9366, Y 35.5257, Z -3.0000, A 0.000, B 0.000, C 0.000 }
gfCNCPoint2[22510] = {X 367.0504, Y 37.5052, Z -3.0000, A 0.000, B 0.000, C 0.000 }
gfCNCPoint2[22511] = {X 365.9927, Y 39.3986, Z -3.0000, A 0.000, B 0.000, C 0.000 }
gfCNCPoint2[22512] = {X 364.7718, Y 41.1911, Z -3.0000, A 0.000, B 0.000, C 0.000 }
gfCNCPoint2[22513] = {X 363.5448, Y 42.7031, Z -3.0000, A 0.000, B 0.000, C 0.000 }
gfCNCPoint2[22514] = {X 362.1899, Y 44.1017, Z -3.0000, A 0.000, B 0.000, C 0.000 }
gfCNCPoint2[22515] = {X 360.7175, Y 45.3761, Z -3.0000, A 0.000, B 0.000, C 0.000 }
gfCNCPoint2[22516] = {X 359.1391, Y 46.5165, Z -3.0000, A 0.000, B 0.000, C 0.000 }
gfCNCPoint2[22517] = {X 357.4668, Y 47.5140, Z -3.0000, A 0.000, B 0.000, C 0.000 }
gfCNCPoint2[22518] = {X 355.5061, Y 48.4045, Z -3.0000, A 0.000, B 0.000, C 0.000 }
gfCNCPoint2[22519] = {X 353.4698, Y 49.1046, Z -3.0000, A 0.000, B 0.000, C 0.000 }
gfCNCPoint2[22520] = {X 351.3761, Y 49.6080, Z -3.0000, A 0.000, B 0.000, C 0.000 }
gfCNCPoint2[22521] = {X 349.2440, Y 49.9101, Z -3.0000, A 0.000, B 0.000, C 0.000 }
gfCNCPoint2[22522] = {X 347.0929, Y 50.0083, Z -3.0000, A 0.000, B 0.000, C 0.000 }
gfCNCPoint2[22523] = {X 345.0263, Y 49.9734, Z -3.0000, A 0.000, B 0.000, C 0.000 }
gfCNCPoint2[22524] = {X 342.9706, Y 49.7594, Z -3.0000, A 0.000, B 0.000, C 0.000 }
gfCNCPoint2[22525] = {X 340.9412, Y 49.3680, Z -3.0000, A 0.000, B 0.000, C 0.000 }
gfCNCPoint2[22526] = {X 338.9534, Y 48.8020, Z -3.0000, A 0.000, B 0.000, C 0.000 }
gfCNCPoint2[22527] = {X 337.0222, Y 48.0657, Z -3.0000, A 0.000, B 0.000, C 0.000 }
gfCNCPoint2[22528] = {X 335.1621, Y 47.1647, Z -3.0000, A 0.000, B 0.000, C 0.000 }
gfCNCPoint2[22529] = {X 333.5781, Y 46.1871, Z -3.0000, A 0.000, B 0.000, C 0.000 }
gfCNCPoint2[22530] = {X 332.0751, Y 45.0890, Z -3.0000, A 0.000, B 0.000, C 0.000 }
gfCNCPoint2[22531] = {X 330.6624, Y 43.8770, Z -3.0000, A 0.000, B 0.000, C 0.000 }
gfCNCPoint2[22532] = {X 329.7214, Y 43.8765, Z -3.0000, A 0.000, B 0.000, C 0.000 }
gfCNCPoint2[22533] = {X 328.8027, Y 43.6721, Z -3.0000, A 0.000, B 0.000, C 0.000 }
gfCNCPoint2[22534] = {X 327.9501, Y 43.2738, Z -3.0000, A 0.000, B 0.000, C 0.000 }
gfCNCPoint2[22535] = {X 327.2040, Y 42.7002, Z -3.0000, A 0.000, B 0.000, C 0.000 }
gfCNCPoint2[22536] = {X 326.5808, Y 42.0925, Z -3.0000, A 0.000, B 0.000, C 0.000 }
gfCNCPoint2[22537] = {X 325.9523, Y 41.3190, Z -3.0000, A 0.000, B 0.000, C 0.000 }
gfCNCPoint2[22538] = {X 325.5179, Y 40.4220, Z -3.0000, A 0.000, B 0.000, C 0.000 }
gfCNCPoint2[22539] = {X 325.3006, Y 39.4493, Z -3.0000, A 0.000, B 0.000, C 0.000 }
gfCNCPoint2[22540] = {X 325.3120, Y 38.4527, Z -3.0000, A 0.000, B 0.000, C 0.000 }
gfCNCPoint2[22541] = {X 325.5514, Y 37.4852, Z -3.0000, A 0.000, B 0.000, C 0.000 }
gfCNCPoint2[22542] = {X 326.0062, Y 36.5984, Z -3.0000, A 0.000, B 0.000, C 0.000 }
gfCNCPoint2[22543] = {X 330.2395, Y 30.2687, Z -3.0000, A 0.000, B 0.000, C 0.000 }
gfCNCPoint2[22544] = {X 330.8409, Y 29.5518, Z -3.0000, A 0.000, B 0.000, C 0.000 }
gfCNCPoint2[22545] = {X 331.5825, Y 28.9812, Z -3.0000, A 0.000, B 0.000, C 0.000 }
gfCNCPoint2[22546] = {X 332.4297, Y 28.5837, Z -3.0000, A 0.000, B 0.000, C 0.000 }
gfCNCPoint2[22547] = {X 333.3425, Y 28.3780, Z -3.0000, A 0.000, B 0.000, C 0.000 }
gfCNCPoint2[22548] = {X 334.2782, Y 28.3736, Z -3.0000, A 0.000, B 0.000, C 0.000 }
gfCNCPoint2[22549] = {X 335.1929, Y 28.5708, Z -3.0000, A 0.000, B 0.000, C 0.000 }
gfCNCPoint2[22550] = {X 336.0437, Y 28.9604, Z -3.0000, A 0.000, B 0.000, C 0.000 }
gfCNCPoint2[22551] = {X 336.7907, Y 29.5240, Z -3.0000, A 0.000, B 0.000, C 0.000 }
gfCNCPoint2[22552] = {X 337.4284, Y 30.1382, Z -3.0000, A 0.000, B 0.000, C 0.000 }
gfCNCPoint2[22553] = {X 337.9530, Y 30.7613, Z -3.0000, A 0.000, B 0.000, C 0.000 }
gfCNCPoint2[22554] = {X 338.3513, Y 31.4717, Z -3.0000, A 0.000, B 0.000, C 0.000 }
gfCNCPoint2[22555] = {X 338.6092, Y 32.2443, Z -3.0000, A 0.000, B 0.000, C 0.000 }
gfCNCPoint2[22556] = {X 338.7175, Y 33.0515, Z -3.0000, A 0.000, B 0.000, C 0.000 }
gfCNCPoint2[22557] = {X 338.6724, Y 33.8647, Z -3.0000, A 0.000, B 0.000, C 0.000 }
gfCNCPoint2[22558] = {X 339.4357, Y 34.5562, Z -3.0000, A 0.000, B 0.000, C 0.000 }
gfCNCPoint2[22559] = {X 340.2331, Y 35.2080, Z -3.0000, A 0.000, B 0.000, C 0.000 }
gfCNCPoint2[22560] = {X 341.5304, Y 36.0602, Z -3.0000, A 0.000, B 0.000, C 0.000 }
gfCNCPoint2[22561] = {X 342.9381, Y 36.7140, Z -3.0000, A 0.000, B 0.000, C 0.000 }
gfCNCPoint2[22562] = {X 344.4261, Y 37.1556, Z -3.0000, A 0.000, B 0.000, C 0.000 }
gfCNCPoint2[22563] = {X 345.9626, Y 37.3755, Z -3.0000, A 0.000, B 0.000, C 0.000 }
gfCNCPoint2[22564] = {X 347.5148, Y 37.3690, Z -3.0000, A 0.000, B 0.000, C 0.000 }
gfCNCPoint2[22565] = {X 348.9555, Y 37.1760, Z -3.0000, A 0.000, B 0.000, C 0.000 }
gfCNCPoint2[22566] = {X 350.3455, Y 36.7510, Z -3.0000, A 0.000, B 0.000, C 0.000 }
gfCNCPoint2[22567] = {X 351.6478, Y 36.1053, Z -3.0000, A 0.000, B 0.000, C 0.000 }
gfCNCPoint2[22568] = {X 352.8276, Y 35.2561, Z -3.0000, A 0.000, B 0.000, C 0.000 }
gfCNCPoint2[22569] = {X 353.9817, Y 34.1352, Z -3.0000, A 0.000, B 0.000, C 0.000 }
gfCNCPoint2[22570] = {X 354.9806, Y 32.8739, Z -3.0000, A 0.000, B 0.000, C 0.000 }
gfCNCPoint2[22571] = {X 355.8072, Y 31.4936, Z -3.0000, A 0.000, B 0.000, C 0.000 }
gfCNCPoint2[22572] = {X 356.4475, Y 30.0177, Z -3.0000, A 0.000, B 0.000, C 0.000 }
gfCNCPoint2[22573] = {X 356.8908, Y 28.4711, Z -3.0000, A 0.000, B 0.000, C 0.000 }
gfCNCPoint2[22574] = {X 357.1641, Y 26.7829, Z -3.0000, A 0.000, B 0.000, C 0.000 }
gfCNCPoint2[22575] = {X 357.2754, Y 25.0763, Z -3.0000, A 0.000, B 0.000, C 0.000 }
gfCNCPoint2[22576] = {X 357.2237, Y 23.3669, Z -3.0000, A 0.000, B 0.000, C 0.000 }
gfCNCPoint2[22577] = {X 357.0095, Y 21.6701, Z -3.0000, A 0.000, B 0.000, C 0.000 }
gfCNCPoint2[22578] = {X 356.6733, Y 20.2206, Z -3.0000, A 0.000, B 0.000, C 0.000 }
gfCNCPoint2[22579] = {X 356.1603, Y 18.8237, Z -3.0000, A 0.000, B 0.000, C 0.000 }
gfCNCPoint2[22580] = {X 355.4783, Y 17.5012, Z -3.0000, A 0.000, B 0.000, C 0.000 }
gfCNCPoint2[22581] = {X 354.6379, Y 16.2732, Z -3.0000, A 0.000, B 0.000, C 0.000 }
gfCNCPoint2[22582] = {X 353.7520, Y 15.2851, Z -3.0000, A 0.000, B 0.000, C 0.000 }
gfCNCPoint2[22583] = {X 352.7336, Y 14.4342, Z -3.0000, A 0.000, B 0.000, C 0.000 }
gfCNCPoint2[22584] = {X 351.6039, Y 13.7379, Z -3.0000, A 0.000, B 0.000, C 0.000 }
gfCNCPoint2[22585] = {X 350.3860, Y 13.2106, Z -3.0000, A 0.000, B 0.000, C 0.000 }
gfCNCPoint2[22586] = {X 349.1052, Y 12.8633, Z -3.0000, A 0.000, B 0.000, C 0.000 }
gfCNCPoint2[22587] = {X 347.3447, Y 12.6444, Z -3.0000, A 0.000, B 0.000, C 0.000 }
gfCNCPoint2[22588] = {X 345.5707, Y 12.6604, Z -3.0000, A 0.000, B 0.000, C 0.000 }
gfCNCPoint2[22589] = {X 343.8144, Y 12.9108, Z -3.0000, A 0.000, B 0.000, C 0.000 }
gfCNCPoint2[22590] = {X 342.1067, Y 13.3914, Z -3.0000, A 0.000, B 0.000, C 0.000 }
gfCNCPoint2[22591] = {X 340.4775, Y 14.0936, Z -3.0000, A 0.000, B 0.000, C 0.000 }
gfCNCPoint2[22592] = {X 338.9555, Y 15.0051, Z -3.0000, A 0.000, B 0.000, C 0.000 }
gfCNCPoint2[22593] = {X 338.9169, Y 15.8497, Z -3.0000, A 0.000, B 0.000, C 0.000 }
gfCNCPoint2[22594] = {X 338.7144, Y 16.6707, Z -3.0000, A 0.000, B 0.000, C 0.000 }
gfCNCPoint2[22595] = {X 338.3559, Y 17.4364, Z -3.0000, A 0.000, B 0.000, C 0.000 }
gfCNCPoint2[22596] = {X 337.8551, Y 18.1177, Z -3.0000, A 0.000, B 0.000, C 0.000 }
gfCNCPoint2[22597] = {X 337.2313, Y 18.6884, Z -3.0000, A 0.000, B 0.000, C 0.000 }
gfCNCPoint2[22598] = {X 336.5140, Y 19.2162, Z -3.0000, A 0.000, B 0.000, C 0.000 }
gfCNCPoint2[22599] = {X 335.6982, Y 19.6754, Z -3.0000, A 0.000, B 0.000, C 0.000 }
gfCNCPoint2[22600] = {X 334.8027, Y 19.9480, Z -3.0000, A 0.000, B 0.000, C 0.000 }
gfCNCPoint2[22601] = {X 333.8694, Y 20.0213, Z -3.0000, A 0.000, B 0.000, C 0.000 }
gfCNCPoint2[22602] = {X 332.9422, Y 19.8919, Z -3.0000, A 0.000, B 0.000, C 0.000 }
gfCNCPoint2[22603] = {X 332.0647, Y 19.5657, Z -3.0000, A 0.000, B 0.000, C 0.000 }
gfCNCPoint2[22604] = {X 331.2781, Y 19.0581, Z -3.0000, A 0.000, B 0.000, C 0.000 }
gfCNCPoint2[22605] = {X 330.6193, Y 18.3931, Z -3.0000, A 0.000, B 0.000, C 0.000 }
gfCNCPoint2[22606] = {X 330.1192, Y 17.6017, Z -3.0000, A 0.000, B 0.000, C 0.000 }
gfCNCPoint2[22607] = {X 326.5942, Y 10.3502, Z -3.0000, A 0.000, B 0.000, C 0.000 }
gfCNCPoint2[22608] = {X 326.2930, Y 9.5271, Z -3.0000, A 0.000, B 0.000, C 0.000 }
gfCNCPoint2[22609] = {X 326.1640, Y 8.6602, Z -3.0000, A 0.000, B 0.000, C 0.000 }
gfCNCPoint2[22610] = {X 326.2128, Y 7.7851, Z -3.0000, A 0.000, B 0.000, C 0.000 }
gfCNCPoint2[22611] = {X 326.4371, Y 6.9378, Z -3.0000, A 0.000, B 0.000, C 0.000 }
gfCNCPoint2[22612] = {X 326.8279, Y 6.1532, Z -3.0000, A 0.000, B 0.000, C 0.000 }
gfCNCPoint2[22613] = {X 327.3690, Y 5.4637, Z -3.0000, A 0.000, B 0.000, C 0.000 }
gfCNCPoint2[22614] = {X 328.0381, Y 4.8976, Z -3.0000, A 0.000, B 0.000, C 0.000 }
gfCNCPoint2[22615] = {X 328.7084, Y 4.4385, Z -3.0000, A 0.000, B 0.000, C 0.000 }
gfCNCPoint2[22616] = {X 329.5889, Y 3.9826, Z -3.0000, A 0.000, B 0.000, C 0.000 }
gfCNCPoint2[22617] = {X 330.5502, Y 3.7394, Z -3.0000, A 0.000, B 0.000, C 0.000 }
gfCNCPoint2[22618] = {X 331.5416, Y 3.7219, Z -3.0000, A 0.000, B 0.000, C 0.000 }
gfCNCPoint2[22619] = {X 332.5110, Y 3.9308, Z -3.0000, A 0.000, B 0.000, C 0.000 }
gfCNCPoint2[22620] = {X 333.9977, Y 3.1012, Z -3.0000, A 0.000, B 0.000, C 0.000 }
gfCNCPoint2[22621] = {X 335.5315, Y 2.3623, Z -3.0000, A 0.000, B 0.000, C 0.000 }
gfCNCPoint2[22622] = {X 337.6677, Y 1.4957, Z -3.0000, A 0.000, B 0.000, C 0.000 }
gfCNCPoint2[22623] = {X 339.8716, Y 0.8196, Z -3.0000, A 0.000, B 0.000, C 0.000 }
gfCNCPoint2[22624] = {X 342.1263, Y 0.3393, Z -3.0000, A 0.000, B 0.000, C 0.000 }
gfCNCPoint2[22625] = {X 344.4144, Y 0.0584, Z -3.0000, A 0.000, B 0.000, C 0.000 }
gfCNCPoint2[22626] = {X 346.7183, Y -0.0209, Z -3.0000, A 0.000, B 0.000, C 0.000 }
gfCNCPoint2[22627] = {X 349.0203, Y 0.1020, Z -3.0000, A 0.000, B 0.000, C 0.000 }
gfCNCPoint2[22628] = {X 351.3026, Y 0.4262, Z -3.0000, A 0.000, B 0.000, C 0.000 }
gfCNCPoint2[22629] = {X 351.5859, Y 0.4787, Z -3.0000, A 0.000, B 0.000, C 0.000 }
gfCNCPoint2[22630] = {X 352.3154, Y -3.4542, Z -3.0000, A 0.000, B 0.000, C 0.000 }
gfCNCPoint2[22631] = {X 351.5713, Y 0.5574, Z -3.0000, A 0.000, B 0.000, C 0.000 }
gfCNCPoint2[22632] = {X 351.8540, Y 0.6098, Z -3.0000, A 0.000, B 0.000, C 0.000 }
gfCNCPoint2[22633] = {X 353.7812, Y 1.0940, Z -3.0000, A 0.000, B 0.000, C 0.000 }
gfCNCPoint2[22634] = {X 355.6539, Y 1.7586, Z -3.0000, A 0.000, B 0.000, C 0.000 }
gfCNCPoint2[22635] = {X 357.4552, Y 2.5977, Z -3.0000, A 0.000, B 0.000, C 0.000 }
gfCNCPoint2[22636] = {X 359.1688, Y 3.6038, Z -3.0000, A 0.000, B 0.000, C 0.000 }
gfCNCPoint2[22637] = {X 360.7794, Y 4.7677, Z -3.0000, A 0.000, B 0.000, C 0.000 }
gfCNCPoint2[22638] = {X 362.2725, Y 6.0790, Z -3.0000, A 0.000, B 0.000, C 0.000 }
gfCNCPoint2[22639] = {X 363.6345, Y 7.5259, Z -3.0000, A 0.000, B 0.000, C 0.000 }
gfCNCPoint2[22640] = {X 365.0970, Y 9.4133, Z -3.0000, A 0.000, B 0.000, C 0.000 }
gfCNCPoint2[22641] = {X 366.3699, Y 11.4333, Z -3.0000, A 0.000, B 0.000, C 0.000 }
gfCNCPoint2[22642] = {X 367.4413, Y 13.5670, Z -3.0000, A 0.000, B 0.000, C 0.000 }
gfCNCPoint2[22643] = {X 368.3011, Y 15.7945, Z -3.0000, A 0.000, B 0.000, C 0.000 }
gfCNCPoint2[22644] = {X 368.9413, Y 18.0947, Z -3.0000, A 0.000, B 0.000, C 0.000 }
gfCNCPoint2[22645] = {X 369.4212, Y 20.7226, Z -3.0000, A 0.000, B 0.000, C 0.000 }
gfCNCPoint2[22646] = {X 369.6771, Y 23.3818, Z -3.0000, A 0.000, B 0.000, C 0.000 }
gfCNCPoint2[22647] = {X 369.7070, Y 26.0530, Z -3.0000, A 0.000, B 0.000, C 0.000 }
gfCNCPoint2[22648] = {X 369.5108, Y 28.7172, Z -3.0000, A 0.000, B 0.000, C 0.000 }
gfCNCPoint2[22649] = {X 369.0899, Y 31.3552, Z -3.0000, A 0.000, B 0.000, C 0.000 }
gfCNCPoint2[22650] = {X 368.5677, Y 33.4530, Z -3.0000, A 0.000, B 0.000, C 0.000 }
gfCNCPoint2[22651] = {X 367.8622, Y 35.4963, Z -3.0000, A 0.000, B 0.000, C 0.000 }
gfCNCPoint2[22652] = {X 366.9788, Y 37.4694, Z -3.0000, A 0.000, B 0.000, C 0.000 }
gfCNCPoint2[22653] = {X 365.9246, Y 39.3566, Z -3.0000, A 0.000, B 0.000, C 0.000 }
gfCNCPoint2[22654] = {X 364.7077, Y 41.1433, Z -3.0000, A 0.000, B 0.000, C 0.000 }
gfCNCPoint2[22655] = {X 363.4851, Y 42.6498, Z -3.0000, A 0.000, B 0.000, C 0.000 }
gfCNCPoint2[22656] = {X 362.1352, Y 44.0433, Z -3.0000, A 0.000, B 0.000, C 0.000 }
gfCNCPoint2[22657] = {X 360.6683, Y 45.3130, Z -3.0000, A 0.000, B 0.000, C 0.000 }
gfCNCPoint2[22658] = {X 359.0957, Y 46.4492, Z -3.0000, A 0.000, B 0.000, C 0.000 }
gfCNCPoint2[22659] = {X 357.4295, Y 47.4432, Z -3.0000, A 0.000, B 0.000, C 0.000 }
gfCNCPoint2[22660] = {X 355.4758, Y 48.3305, Z -3.0000, A 0.000, B 0.000, C 0.000 }
gfCNCPoint2[22661] = {X 353.4465, Y 49.0281, Z -3.0000, A 0.000, B 0.000, C 0.000 }
gfCNCPoint2[22662] = {X 351.3601, Y 49.5296, Z -3.0000, A 0.000, B 0.000, C 0.000 }
gfCNCPoint2[22663] = {X 349.2355, Y 49.8306, Z -3.0000, A 0.000, B 0.000, C 0.000 }
gfCNCPoint2[22664] = {X 347.0919, Y 49.9283, Z -3.0000, A 0.000, B 0.000, C 0.000 }
gfCNCPoint2[22665] = {X 345.0322, Y 49.8936, Z -3.0000, A 0.000, B 0.000, C 0.000 }
gfCNCPoint2[22666] = {X 342.9834, Y 49.6805, Z -3.0000, A 0.000, B 0.000, C 0.000 }
gfCNCPoint2[22667] = {X 340.9607, Y 49.2904, Z -3.0000, A 0.000, B 0.000, C 0.000 }
gfCNCPoint2[22668] = {X 338.9795, Y 48.7263, Z -3.0000, A 0.000, B 0.000, C 0.000 }
gfCNCPoint2[22669] = {X 337.0547, Y 47.9926, Z -3.0000, A 0.000, B 0.000, C 0.000 }
gfCNCPoint2[22670] = {X 335.2007, Y 47.0946, Z -3.0000, A 0.000, B 0.000, C 0.000 }
gfCNCPoint2[22671] = {X 333.6121, Y 46.1136, Z -3.0000, A 0.000, B 0.000, C 0.000 }
gfCNCPoint2[22672] = {X 332.1054, Y 45.0109, Z -3.0000, A 0.000, B 0.000, C 0.000 }
gfCNCPoint2[22673] = {X 330.6900, Y 43.7933, Z -3.0000, A 0.000, B 0.000, C 0.000 }
gfCNCPoint2[22674] = {X 329.7573, Y 43.7998, Z -3.0000, A 0.000, B 0.000, C 0.000 }
gfCNCPoint2[22675] = {X 328.8457, Y 43.6022, Z -3.0000, A 0.000, B 0.000, C 0.000 }
gfCNCPoint2[22676] = {X 327.9995, Y 43.2101, Z -3.0000, A 0.000, B 0.000, C 0.000 }
gfCNCPoint2[22677] = {X 327.2594, Y 42.6425, Z -3.0000, A 0.000, B 0.000, C 0.000 }
gfCNCPoint2[22678] = {X 326.6366, Y 42.0352, Z -3.0000, A 0.000, B 0.000, C 0.000 }
gfCNCPoint2[22679] = {X 326.0198, Y 41.2760, Z -3.0000, A 0.000, B 0.000, C 0.000 }
gfCNCPoint2[22680] = {X 325.5934, Y 40.3956, Z -3.0000, A 0.000, B 0.000, C 0.000 }
gfCNCPoint2[22681] = {X 325.3802, Y 39.4410, Z -3.0000, A 0.000, B 0.000, C 0.000 }
gfCNCPoint2[22682] = {X 325.3913, Y 38.4628, Z -3.0000, A 0.000, B 0.000, C 0.000 }
gfCNCPoint2[22683] = {X 325.6264, Y 37.5133, Z -3.0000, A 0.000, B 0.000, C 0.000 }
gfCNCPoint2[22684] = {X 326.0727, Y 36.6429, Z -3.0000, A 0.000, B 0.000, C 0.000 }
gfCNCPoint2[22685] = {X 330.3060, Y 30.3132, Z -3.0000, A 0.000, B 0.000, C 0.000 }
gfCNCPoint2[22686] = {X 330.8963, Y 29.6096, Z -3.0000, A 0.000, B 0.000, C 0.000 }
gfCNCPoint2[22687] = {X 331.6242, Y 29.0496, Z -3.0000, A 0.000, B 0.000, C 0.000 }
gfCNCPoint2[22688] = {X 332.4556, Y 28.6594, Z -3.0000, A 0.000, B 0.000, C 0.000 }
gfCNCPoint2[22689] = {X 333.3515, Y 28.4575, Z -3.0000, A 0.000, B 0.000, C 0.000 }
gfCNCPoint2[22690] = {X 334.2699, Y 28.4532, Z -3.0000, A 0.000, B 0.000, C 0.000 }
gfCNCPoint2[22691] = {X 335.1677, Y 28.6467, Z -3.0000, A 0.000, B 0.000, C 0.000 }
gfCNCPoint2[22692] = {X 336.0027, Y 29.0291, Z -3.0000, A 0.000, B 0.000, C 0.000 }
gfCNCPoint2[22693] = {X 336.7358, Y 29.5823, Z -3.0000, A 0.000, B 0.000, C 0.000 }
gfCNCPoint2[22694] = {X 337.3723, Y 30.1953, Z -3.0000, A 0.000, B 0.000, C 0.000 }
gfCNCPoint2[22695] = {X 337.8919, Y 30.8136, Z -3.0000, A 0.000, B 0.000, C 0.000 }
gfCNCPoint2[22696] = {X 338.2848, Y 31.5192, Z -3.0000, A 0.000, B 0.000, C 0.000 }
gfCNCPoint2[22697] = {X 338.5368, Y 32.2865, Z -3.0000, A 0.000, B 0.000, C 0.000 }
gfCNCPoint2[22698] = {X 338.6388, Y 33.0877, Z -3.0000, A 0.000, B 0.000, C 0.000 }
gfCNCPoint2[22699] = {X 338.5869, Y 33.8937, Z -3.0000, A 0.000, B 0.000, C 0.000 }
gfCNCPoint2[22700] = {X 339.3677, Y 34.6032, Z -3.0000, A 0.000, B 0.000, C 0.000 }
gfCNCPoint2[22701] = {X 340.1842, Y 35.2714, Z -3.0000, A 0.000, B 0.000, C 0.000 }
gfCNCPoint2[22702] = {X 341.4911, Y 36.1299, Z -3.0000, A 0.000, B 0.000, C 0.000 }
gfCNCPoint2[22703] = {X 342.9093, Y 36.7887, Z -3.0000, A 0.000, B 0.000, C 0.000 }
gfCNCPoint2[22704] = {X 344.4083, Y 37.2336, Z -3.0000, A 0.000, B 0.000, C 0.000 }
gfCNCPoint2[22705] = {X 345.9562, Y 37.4552, Z -3.0000, A 0.000, B 0.000, C 0.000 }
gfCNCPoint2[22706] = {X 347.5199, Y 37.4488, Z -3.0000, A 0.000, B 0.000, C 0.000 }
gfCNCPoint2[22707] = {X 348.9733, Y 37.2540, Z -3.0000, A 0.000, B 0.000, C 0.000 }
gfCNCPoint2[22708] = {X 350.3756, Y 36.8251, Z -3.0000, A 0.000, B 0.000, C 0.000 }
gfCNCPoint2[22709] = {X 351.6893, Y 36.1737, Z -3.0000, A 0.000, B 0.000, C 0.000 }
gfCNCPoint2[22710] = {X 352.8795, Y 35.3170, Z -3.0000, A 0.000, B 0.000, C 0.000 }
gfCNCPoint2[22711] = {X 354.0411, Y 34.1888, Z -3.0000, A 0.000, B 0.000, C 0.000 }
gfCNCPoint2[22712] = {X 355.0464, Y 32.9193, Z -3.0000, A 0.000, B 0.000, C 0.000 }
gfCNCPoint2[22713] = {X 355.8784, Y 31.5300, Z -3.0000, A 0.000, B 0.000, C 0.000 }
gfCNCPoint2[22714] = {X 356.5229, Y 30.0445, Z -3.0000, A 0.000, B 0.000, C 0.000 }
gfCNCPoint2[22715] = {X 356.9690, Y 28.4878, Z -3.0000, A 0.000, B 0.000, C 0.000 }
gfCNCPoint2[22716] = {X 357.2436, Y 26.7920, Z -3.0000, A 0.000, B 0.000, C 0.000 }
gfCNCPoint2[22717] = {X 357.3554, Y 25.0778, Z -3.0000, A 0.000, B 0.000, C 0.000 }
gfCNCPoint2[22718] = {X 357.3035, Y 23.3607, Z -3.0000, A 0.000, B 0.000, C 0.000 }
gfCNCPoint2[22719] = {X 357.0883, Y 21.6563, Z -3.0000, A 0.000, B 0.000, C 0.000 }
gfCNCPoint2[22720] = {X 356.7499, Y 20.1973, Z -3.0000, A 0.000, B 0.000, C 0.000 }
gfCNCPoint2[22721] = {X 356.2334, Y 18.7913, Z -3.0000, A 0.000, B 0.000, C 0.000 }
gfCNCPoint2[22722] = {X 355.5469, Y 17.4600, Z -3.0000, A 0.000, B 0.000, C 0.000 }
gfCNCPoint2[22723] = {X 354.7010, Y 16.2240, Z -3.0000, A 0.000, B 0.000, C 0.000 }
gfCNCPoint2[22724] = {X 353.8074, Y 15.2274, Z -3.0000, A 0.000, B 0.000, C 0.000 }
gfCNCPoint2[22725] = {X 352.7802, Y 14.3691, Z -3.0000, A 0.000, B 0.000, C 0.000 }
gfCNCPoint2[22726] = {X 351.6407, Y 13.6669, Z -3.0000, A 0.000, B 0.000, C 0.000 }
gfCNCPoint2[22727] = {X 350.4124, Y 13.1351, Z -3.0000, A 0.000, B 0.000, C 0.000 }
gfCNCPoint2[22728] = {X 349.1205, Y 12.7848, Z -3.0000, A 0.000, B 0.000, C 0.000 }
gfCNCPoint2[22729] = {X 347.3419, Y 12.5642, Z -3.0000, A 0.000, B 0.000, C 0.000 }
gfCNCPoint2[22730] = {X 345.5499, Y 12.5817, Z -3.0000, A 0.000, B 0.000, C 0.000 }
gfCNCPoint2[22731] = {X 343.7760, Y 12.8372, Z -3.0000, A 0.000, B 0.000, C 0.000 }
gfCNCPoint2[22732] = {X 342.0518, Y 13.3260, Z -3.0000, A 0.000, B 0.000, C 0.000 }
gfCNCPoint2[22733] = {X 340.4078, Y 14.0395, Z -3.0000, A 0.000, B 0.000, C 0.000 }
gfCNCPoint2[22734] = {X 338.8731, Y 14.9650, Z -3.0000, A 0.000, B 0.000, C 0.000 }
gfCNCPoint2[22735] = {X 338.8426, Y 15.8031, Z -3.0000, A 0.000, B 0.000, C 0.000 }
gfCNCPoint2[22736] = {X 338.6478, Y 16.6189, Z -3.0000, A 0.000, B 0.000, C 0.000 }
gfCNCPoint2[22737] = {X 338.2962, Y 17.3803, Z -3.0000, A 0.000, B 0.000, C 0.000 }
gfCNCPoint2[22738] = {X 337.8015, Y 18.0577, Z -3.0000, A 0.000, B 0.000, C 0.000 }
gfCNCPoint2[22739] = {X 337.1833, Y 18.6244, Z -3.0000, A 0.000, B 0.000, C 0.000 }
gfCNCPoint2[22740] = {X 336.4675, Y 19.1512, Z -3.0000, A 0.000, B 0.000, C 0.000 }
gfCNCPoint2[22741] = {X 335.6668, Y 19.6018, Z -3.0000, A 0.000, B 0.000, C 0.000 }
gfCNCPoint2[22742] = {X 334.7878, Y 19.8694, Z -3.0000, A 0.000, B 0.000, C 0.000 }
gfCNCPoint2[22743] = {X 333.8718, Y 19.9414, Z -3.0000, A 0.000, B 0.000, C 0.000 }
gfCNCPoint2[22744] = {X 332.9618, Y 19.8143, Z -3.0000, A 0.000, B 0.000, C 0.000 }
gfCNCPoint2[22745] = {X 332.1006, Y 19.4942, Z -3.0000, A 0.000, B 0.000, C 0.000 }
gfCNCPoint2[22746] = {X 331.3285, Y 18.9960, Z -3.0000, A 0.000, B 0.000, C 0.000 }
gfCNCPoint2[22747] = {X 330.6819, Y 18.3433, Z -3.0000, A 0.000, B 0.000, C 0.000 }
gfCNCPoint2[22748] = {X 330.1911, Y 17.5665, Z -3.0000, A 0.000, B 0.000, C 0.000 }
gfCNCPoint2[22749] = {X 326.6662, Y 10.3152, Z -3.0000, A 0.000, B 0.000, C 0.000 }
gfCNCPoint2[22750] = {X 326.3374, Y 9.3676, Z -3.0000, A 0.000, B 0.000, C 0.000 }
gfCNCPoint2[22751] = {X 326.2405, Y 8.3693, Z -3.0000, A 0.000, B 0.000, C 0.000 }
gfCNCPoint2[22752] = {X 326.3807, Y 7.3762, Z -3.0000, A 0.000, B 0.000, C 0.000 }
gfCNCPoint2[22753] = {X 326.7504, Y 6.4438, Z -3.0000, A 0.000, B 0.000, C 0.000 }
gfCNCPoint2[22754] = {X 327.3287, Y 5.6243, Z -3.0000, A 0.000, B 0.000, C 0.000 }
gfCNCPoint2[22755] = {X 328.0833, Y 4.9636, Z -3.0000, A 0.000, B 0.000, C 0.000 }
gfCNCPoint2[22756] = {X 328.7533, Y 4.5047, Z -3.0000, A 0.000, B 0.000, C 0.000 }
gfCNCPoint2[22757] = {X 329.6262, Y 4.0540, Z -3.0000, A 0.000, B 0.000, C 0.000 }
gfCNCPoint2[22758] = {X 330.5793, Y 3.8163, Z -3.0000, A 0.000, B 0.000, C 0.000 }
gfCNCPoint2[22759] = {X 331.5615, Y 3.8043, Z -3.0000, A 0.000, B 0.000, C 0.000 }
gfCNCPoint2[22760] = {X 332.5201, Y 4.0186, Z -3.0000, A 0.000, B 0.000, C 0.000 }
gfCNCPoint2[22761] = {X 334.0183, Y 3.1806, Z -3.0000, A 0.000, B 0.000, C 0.000 }
gfCNCPoint2[22762] = {X 335.5645, Y 2.4352, Z -3.0000, A 0.000, B 0.000, C 0.000 }
gfCNCPoint2[22763] = {X 337.6942, Y 1.5712, Z -3.0000, A 0.000, B 0.000, C 0.000 }
gfCNCPoint2[22764] = {X 339.8914, Y 0.8971, Z -3.0000, A 0.000, B 0.000, C 0.000 }
gfCNCPoint2[22765] = {X 342.1393, Y 0.4182, Z -3.0000, A 0.000, B 0.000, C 0.000 }
gfCNCPoint2[22766] = {X 344.4205, Y 0.1382, Z -3.0000, A 0.000, B 0.000, C 0.000 }
gfCNCPoint2[22767] = {X 346.7174, Y 0.0591, Z -3.0000, A 0.000, B 0.000, C 0.000 }
gfCNCPoint2[22768] = {X 349.0125, Y 0.1816, Z -3.0000, A 0.000, B 0.000, C 0.000 }
gfCNCPoint2[22769] = {X 351.2879, Y 0.5048, Z -3.0000, A 0.000, B 0.000, C 0.000 }
gfCNCPoint2[22770] = {X 351.5713, Y 0.5574, Z -3.0000, A 0.000, B 0.000, C 0.000 }
gfCNCPoint2[22771] = {X 352.3008, Y -3.3756, Z -3.0000, A 0.000, B 0.000, C 0.000 }
gfCNCPoint2[22772] = {X 351.5567, Y 0.6360, Z -3.0000, A 0.000, B 0.000, C 0.000 }
gfCNCPoint2[22773] = {X 351.8388, Y 0.6883, Z -3.0000, A 0.000, B 0.000, C 0.000 }
gfCNCPoint2[22774] = {X 353.7586, Y 1.1707, Z -3.0000, A 0.000, B 0.000, C 0.000 }
gfCNCPoint2[22775] = {X 355.6240, Y 1.8328, Z -3.0000, A 0.000, B 0.000, C 0.000 }
gfCNCPoint2[22776] = {X 357.4183, Y 2.6687, Z -3.0000, A 0.000, B 0.000, C 0.000 }
gfCNCPoint2[22777] = {X 359.1253, Y 3.6709, Z -3.0000, A 0.000, B 0.000, C 0.000 }
gfCNCPoint2[22778] = {X 360.7297, Y 4.8304, Z -3.0000, A 0.000, B 0.000, C 0.000 }
gfCNCPoint2[22779] = {X 362.2169, Y 6.1366, Z -3.0000, A 0.000, B 0.000, C 0.000 }
gfCNCPoint2[22780] = {X 363.5737, Y 7.5779, Z -3.0000, A 0.000, B 0.000, C 0.000 }
gfCNCPoint2[22781] = {X 365.0314, Y 9.4591, Z -3.0000, A 0.000, B 0.000, C 0.000 }
gfCNCPoint2[22782] = {X 366.3002, Y 11.4726, Z -3.0000, A 0.000, B 0.000, C 0.000 }
gfCNCPoint2[22783] = {X 367.3681, Y 13.5994, Z -3.0000, A 0.000, B 0.000, C 0.000 }
gfCNCPoint2[22784] = {X 368.2252, Y 15.8196, Z -3.0000, A 0.000, B 0.000, C 0.000 }
gfCNCPoint2[22785] = {X 368.8633, Y 18.1124, Z -3.0000, A 0.000, B 0.000, C 0.000 }
gfCNCPoint2[22786] = {X 369.3420, Y 20.7337, Z -3.0000, A 0.000, B 0.000, C 0.000 }
gfCNCPoint2[22787] = {X 369.5972, Y 23.3860, Z -3.0000, A 0.000, B 0.000, C 0.000 }
gfCNCPoint2[22788] = {X 369.6271, Y 26.0505, Z -3.0000, A 0.000, B 0.000, C 0.000 }
gfCNCPoint2[22789] = {X 369.4314, Y 28.7079, Z -3.0000, A 0.000, B 0.000, C 0.000 }
gfCNCPoint2[22790] = {X 369.0115, Y 31.3393, Z -3.0000, A 0.000, B 0.000, C 0.000 }
gfCNCPoint2[22791] = {X 368.4910, Y 33.4302, Z -3.0000, A 0.000, B 0.000, C 0.000 }
gfCNCPoint2[22792] = {X 367.7878, Y 35.4669, Z -3.0000, A 0.000, B 0.000, C 0.000 }
gfCNCPoint2[22793] = {X 366.9073, Y 37.4335, Z -3.0000, A 0.000, B 0.000, C 0.000 }
gfCNCPoint2[22794] = {X 365.8565, Y 39.3146, Z -3.0000, A 0.000, B 0.000, C 0.000 }
gfCNCPoint2[22795] = {X 364.6435, Y 41.0955, Z -3.0000, A 0.000, B 0.000, C 0.000 }
